LIN {X 0,Y 481.085,Z 509.859,A -85,B 0,C 180,E1 -6735.62,E2 -6735.62} C_VEL
LIN {X 0,Y 481.237,Z 504.412,A -85,B 0,C 180,E1 -6738.202,E2 -6738.202} C_VEL
LIN {X 0,Y 481.286,Z 497.171,A -85,B 0,C 180,E1 -6741.603,E2 -6741.603} C_VEL
LIN {X 0,Y 481.313,Z 491.765,A -85,B 0,C 180,E1 -6744.133,E2 -6744.133} C_VEL
LIN {X 0,Y 481.415,Z 488.11,A -85,B 0,C 180,E1 -6745.814,E2 -6745.814} C_VEL
LIN {X 0,Y 481.345,Z 485.341,A -85,B 0,C 180,E1 -6747.175,E2 -6747.175} C_VEL
LIN {X 0,Y 481.839,Z 485.279,A -85,B 0,C 180,E1 -6749.164,E2 -6749.164} C_VEL
LIN {X 0,Y 481.908,Z 485.27,A -85,B 0,C 180,E1 -6750.835,E2 -6750.835} C_VEL
LIN {X 0,Y 481.93,Z 485.268,A -85,B 0,C 180,E1 -6752.507,E2 -6752.507} C_VEL
LIN {X 0,Y 481.82,Z 485.281,A -85,B 0,C 180,E1 -6755.86,E2 -6755.86} C_VEL
LIN {X 0,Y 481.763,Z 485.289,A -85,B 0,C 180,E1 -6758.388,E2 -6758.388} C_VEL
LIN {X 0,Y 481.752,Z 485.289,A -85,B 0,C 180,E1 -6761.784,E2 -6761.784} C_VEL
LIN {X 0,Y 481.745,Z 485.289,A -85,B 0,C 180,E1 -6765.224,E2 -6765.224} C_VEL
LIN {X 0,Y 481.713,Z 485.294,A -85,B 0,C 180,E1 -6768.721,E2 -6768.721} C_VEL
LIN {X 0,Y 481.648,Z 485.301,A -85,B 0,C 180,E1 -6771.394,E2 -6771.394} C_VEL
LIN {X 0,Y 481.678,Z 485.301,A -85,B 0,C 180,E1 -6774.113,E2 -6774.113} C_VEL
LIN {X 0,Y 481.752,Z 485.288,A -85,B 0,C 180,E1 -6777.14,E2 -6777.14} C_VEL
LIN {X 0,Y 481.688,Z 485.297,A -85,B 0,C 180,E1 -6779.74,E2 -6779.74} C_VEL
LIN {X 0,Y 481.673,Z 485.299,A -85,B 0,C 180,E1 -6782.674,E2 -6782.674} C_VEL
LIN {X 0,Y 481.643,Z 485.303,A -85,B 0,C 180,E1 -6785.708,E2 -6785.708} C_VEL
LIN {X 0,Y 481.67,Z 485.298,A -85,B 0,C 180,E1 -6788.859,E2 -6788.859} C_VEL
LIN {X 0,Y 481.661,Z 485.303,A -85,B 0,C 180,E1 -6791.914,E2 -6791.914} C_VEL
LIN {X 0,Y 481.659,Z 485.301,A -85,B 0,C 180,E1 -6794.457,E2 -6794.457} C_VEL
LIN {X 0,Y 481.687,Z 485.297,A -85,B 0,C 180,E1 -6796.845,E2 -6796.845} C_VEL
LIN {X 0,Y 481.688,Z 485.3,A -85,B 0,C 180,E1 -6800.061,E2 -6800.061} C_VEL
LIN {X 0,Y 481.624,Z 485.304,A -85,B 0,C 180,E1 -6803.253,E2 -6803.253} C_VEL
LIN {X 0,Y 481.707,Z 485.295,A -85,B 0,C 180,E1 -6806.33,E2 -6806.33} C_VEL
LIN {X 0,Y 481.649,Z 485.302,A -85,B 0,C 180,E1 -6809.417,E2 -6809.417} C_VEL
LIN {X 0,Y 481.7,Z 485.297,A -85,B 0,C 180,E1 -6812.168,E2 -6812.168} C_VEL
LIN {X 0,Y 481.717,Z 485.292,A -85,B 0,C 180,E1 -6814.97,E2 -6814.97} C_VEL
LIN {X 0,Y 481.651,Z 485.303,A -85,B 0,C 180,E1 -6817.705,E2 -6817.705} C_VEL
LIN {X 0,Y 481.706,Z 485.295,A -85,B 0,C 180,E1 -6820.393,E2 -6820.393} C_VEL
LIN {X 0,Y 481.689,Z 485.297,A -85,B 0,C 180,E1 -6823.034,E2 -6823.034} C_VEL
LIN {X 0,Y 481.688,Z 485.298,A -85,B 0,C 180,E1 -6825.639,E2 -6825.639} C_VEL
LIN {X 0,Y 481.793,Z 485.286,A -85,B 0,C 180,E1 -6828.216,E2 -6828.216} C_VEL
LIN {X 0,Y 481.761,Z 485.289,A -85,B 0,C 180,E1 -6831.612,E2 -6831.612} C_VEL
LIN {X 0,Y 481.814,Z 485.283,A -85,B 0,C 180,E1 -6834.139,E2 -6834.139} C_VEL
LIN {X 0,Y 481.928,Z 485.268,A -85,B 0,C 180,E1 -6837.492,E2 -6837.492} C_VEL
LIN {X 0,Y 481.939,Z 485.267,A -85,B 0,C 180,E1 -6840,E2 -6840} C_VEL
LIN {X 0,Y 481.926,Z 485.268,A -85,B 0,C 180,E1 -6842.507,E2 -6842.507} C_VEL
LIN {X 0,Y 481.816,Z 485.283,A -85,B 0,C 180,E1 -6845.86,E2 -6845.86} C_VEL
LIN {X 0,Y 481.761,Z 485.289,A -85,B 0,C 180,E1 -6848.388,E2 -6848.388} C_VEL
LIN {X 0,Y 481.749,Z 485.291,A -85,B 0,C 180,E1 -6851.785,E2 -6851.785} C_VEL
LIN {X 0,Y 481.74,Z 485.291,A -85,B 0,C 180,E1 -6855.224,E2 -6855.224} C_VEL
LIN {X 0,Y 481.71,Z 485.293,A -85,B 0,C 180,E1 -6858.722,E2 -6858.722} C_VEL
LIN {X 0,Y 481.645,Z 485.304,A -85,B 0,C 180,E1 -6861.395,E2 -6861.395} C_VEL
LIN {X 0,Y 481.675,Z 485.299,A -85,B 0,C 180,E1 -6864.113,E2 -6864.113} C_VEL
LIN {X 0,Y 481.744,Z 485.29,A -85,B 0,C 180,E1 -6867.139,E2 -6867.139} C_VEL
LIN {X 0,Y 481.686,Z 485.3,A -85,B 0,C 180,E1 -6869.741,E2 -6869.741} C_VEL
LIN {X 0,Y 481.671,Z 485.299,A -85,B 0,C 180,E1 -6872.674,E2 -6872.674} C_VEL
LIN {X 0,Y 481.641,Z 485.306,A -85,B 0,C 180,E1 -6875.709,E2 -6875.709} C_VEL
LIN {X 0,Y 481.668,Z 485.299,A -85,B 0,C 180,E1 -6878.859,E2 -6878.859} C_VEL
LIN {X 0,Y 481.66,Z 485.301,A -85,B 0,C 180,E1 -6881.914,E2 -6881.914} C_VEL
LIN {X 0,Y 481.658,Z 485.3,A -85,B 0,C 180,E1 -6884.457,E2 -6884.457} C_VEL
LIN {X 0,Y 481.647,Z 485.303,A -85,B 0,C 180,E1 -6887.84,E2 -6887.84} C_VEL
LIN {X 0,Y 481.718,Z 485.292,A -85,B 0,C 180,E1 -6890.646,E2 -6890.646} C_VEL
LIN {X 0,Y 481.642,Z 485.305,A -85,B 0,C 180,E1 -6894.291,E2 -6894.291} C_VEL
LIN {X 0,Y 481.734,Z 485.411,A -85,B 0,C 180,E1 -6895.75,E2 -6895.75} C_VEL
LIN {X 0,Y 482.859,Z 492.268,A -85,B 0,C 180,E1 -6898.401,E2 -6898.401} C_VEL
LIN {X 0,Y 482.63,Z 499.151,A -85,B 0,C 180,E1 -6900.893,E2 -6900.893} C_VEL
LIN {X 0,Y 482.277,Z 506.878,A -85,B 0,C 180,E1 -6903.612,E2 -6903.612} C_VEL
LIN {X 0,Y 481.947,Z 514.883,A -85,B 0,C 180,E1 -6906.359,E2 -6906.359} C_VEL
LIN {X 0,Y 481.668,Z 524.244,A -85,B 0,C 180,E1 -6909.502,E2 -6909.502} C_VEL
LIN {X 0,Y 481.4,Z 533.634,A -85,B 0,C 180,E1 -6912.586,E2 -6912.586} C_VEL
LIN {X 0,Y 481.187,Z 543.054,A -85,B 0,C 180,E1 -6915.624,E2 -6915.624} C_VEL
LIN {X 0,Y 481.103,Z 551.174,A -85,B 0,C 180,E1 -6918.228,E2 -6918.228} C_VEL
LIN {X 0,Y 482.499,Z 564.801,A -85,B 0,C 180,E1 -6918.713,E2 -6918.713} C_VEL
LIN {X 0,Y 482.362,Z 574.583,A -85,B 0,C 180,E1 -6919.188,E2 -6919.188} C_VEL
LIN {X 0,Y 482.16,Z 583.023,A -85,B 0,C 180,E1 -6919.715,E2 -6919.715} C_VEL
LIN {X 0,Y 481.922,Z 591.176,A -85,B 0,C 180,E1 -6920.346,E2 -6920.346} C_VEL
LIN {X 0,Y 481.622,Z 598.943,A -85,B 0,C 180,E1 -6921.081,E2 -6921.081} C_VEL
LIN {X 0,Y 481.355,Z 607.096,A -85,B 0,C 180,E1 -6922.028,E2 -6922.028} C_VEL
LIN {X 0,Y 481.168,Z 614.279,A -85,B 0,C 180,E1 -6923.079,E2 -6923.079} C_VEL
LIN {X 0,Y 481.055,Z 619.93,A -85,B 0,C 180,E1 -6924.131,E2 -6924.131} C_VEL
LIN {X 0,Y 480.885,Z 625.177,A -85,B 0,C 180,E1 -6925.39,E2 -6925.39} C_VEL
LIN {X 0,Y 480.937,Z 627.877,A -85,B 0,C 180,E1 -6926.23,E2 -6926.23} C_VEL
LIN {X 0,Y 480.848,Z 630.817,A -85,B 0,C 180,E1 -6927.487,E2 -6927.487} C_VEL
LIN {X 0,Y 480.822,Z 632.089,A -85,B 0,C 180,E1 -6928.325,E2 -6928.325} C_VEL
LIN {X 0,Y 480.758,Z 632.873,A -85,B 0,C 180,E1 -6929.163,E2 -6929.163} C_VEL
LIN {X 0,Y 480.74,Z 633.154,A -85,B 0,C 180,E1 -6930,E2 -6930} C_VEL
LIN {X 0,Y 480.758,Z 632.838,A -85,B 0,C 180,E1 -6930.838,E2 -6930.838} C_VEL
LIN {X 0,Y 480.822,Z 632.029,A -85,B 0,C 180,E1 -6931.676,E2 -6931.676} C_VEL
LIN {X 0,Y 480.849,Z 630.732,A -85,B 0,C 180,E1 -6932.514,E2 -6932.514} C_VEL
LIN {X 0,Y 480.94,Z 627.734,A -85,B 0,C 180,E1 -6933.771,E2 -6933.771} C_VEL
LIN {X 0,Y 480.885,Z 624.999,A -85,B 0,C 180,E1 -6934.611,E2 -6934.611} C_VEL
LIN {X 0,Y 481.057,Z 619.674,A -85,B 0,C 180,E1 -6935.87,E2 -6935.87} C_VEL
LIN {X 0,Y 481.209,Z 612.625,A -85,B 0,C 180,E1 -6937.132,E2 -6937.132} C_VEL
LIN {X 0,Y 481.403,Z 604.966,A -85,B 0,C 180,E1 -6938.184,E2 -6938.184} C_VEL
LIN {X 0,Y 481.621,Z 598.453,A -85,B 0,C 180,E1 -6938.92,E2 -6938.92} C_VEL
LIN {X 0,Y 481.882,Z 590.591,A -85,B 0,C 180,E1 -6939.656,E2 -6939.656} C_VEL
LIN {X 0,Y 482.097,Z 582.346,A -85,B 0,C 180,E1 -6940.287,E2 -6940.287} C_VEL
LIN {X 0,Y 482.403,Z 571.991,A -85,B 0,C 180,E1 -6940.918,E2 -6940.918} C_VEL
LIN {X 0,Y 482.382,Z 564.502,A -85,B 0,C 180,E1 -6941.267,E2 -6941.267} C_VEL
LIN {X 0,Y 481.115,Z 552.246,A -85,B 0,C 180,E1 -6941.715,E2 -6941.715} C_VEL
LIN {X 0,Y 481.004,Z 550.841,A -85,B 0,C 180,E1 -6941.75,E2 -6941.75} C_VEL
LIN {X 0,Y 481.17,Z 540.308,A -85,B 0,C 180,E1 -6945.243,E2 -6945.243} C_VEL
LIN {X 0,Y 481.361,Z 530.012,A -85,B 0,C 180,E1 -6948.736,E2 -6948.736} C_VEL
LIN {X 0,Y 481.539,Z 521.127,A -85,B 0,C 180,E1 -6951.85,E2 -6951.85} C_VEL
LIN {X 0,Y 481.787,Z 513.681,A -85,B 0,C 180,E1 -6954.566,E2 -6954.566} C_VEL
LIN {X 0,Y 482.085,Z 506.773,A -85,B 0,C 180,E1 -6957.217,E2 -6957.217} C_VEL
LIN {X 0,Y 482.519,Z 499.627,A -85,B 0,C 180,E1 -6960.166,E2 -6960.166} C_VEL
LIN {X 0,Y 482.874,Z 494.307,A -85,B 0,C 180,E1 -6962.583,E2 -6962.583} C_VEL
LIN {X 0,Y 482.76,Z 491.673,A -85,B 0,C 180,E1 -6963.922,E2 -6963.922} C_VEL
LIN {X 0,Y 481.959,Z 486.988,A -85,B 0,C 180,E1 -6966.718,E2 -6966.718} C_VEL
LIN {X 0,Y 481.658,Z 485.303,A -85,B 0,C 180,E1 -6968.008,E2 -6968.008} C_VEL
LIN {X 0,Y 481.659,Z 485.302,A -85,B 0,C 180,E1 -6971.042,E2 -6971.042} C_VEL
LIN {X 0,Y 481.662,Z 485.301,A -85,B 0,C 180,E1 -6974.458,E2 -6974.458} C_VEL
LIN {X 0,Y 481.656,Z 485.302,A -85,B 0,C 180,E1 -6977.84,E2 -6977.84} C_VEL
LIN {X 0,Y 481.683,Z 485.299,A -85,B 0,C 180,E1 -6980.651,E2 -6980.651} C_VEL
LIN {X 0,Y 481.63,Z 485.307,A -85,B 0,C 180,E1 -6983.376,E2 -6983.376} C_VEL
LIN {X 0,Y 481.672,Z 485.303,A -85,B 0,C 180,E1 -6986.327,E2 -6986.327} C_VEL
LIN {X 0,Y 481.625,Z 485.502,A -85,B 0,C 180,E1 -6987.322,E2 -6987.322} C_VEL
LIN {X 0,Y 481.574,Z 488.341,A -85,B 0,C 180,E1 -6990.252,E2 -6990.252} C_VEL
LIN {X 0,Y 481.43,Z 491.329,A -85,B 0,C 180,E1 -6993.093,E2 -6993.093} C_VEL
LIN {X 0,Y 481.283,Z 494.419,A -85,B 0,C 180,E1 -6995.866,E2 -6995.866} C_VEL
LIN {X 0,Y 481.208,Z 498.618,A -85,B 0,C 180,E1 -6999.481,E2 -6999.481} C_VEL
LIN {X 0,Y 481.075,Z 501.825,A -85,B 0,C 180,E1 -7002.134,E2 -7002.134} C_VEL
LIN {X 0,Y 481.082,Z 505.064,A -85,B 0,C 180,E1 -7004.754,E2 -7004.754} C_VEL
LIN {X 0,Y 481.019,Z 509.748,A -85,B 0,C 180,E1 -7008.382,E2 -7008.382} C_VEL
LIN {X 0,Y 482.651,Z 519.951,A -85,B 0,C 180,E1 -7008.796,E2 -7008.796} C_VEL
LIN {X 0,Y 482.57,Z 529.986,A -85,B 0,C 180,E1 -7009.299,E2 -7009.299} C_VEL
LIN {X 0,Y 482.326,Z 538.199,A -85,B 0,C 180,E1 -7009.824,E2 -7009.824} C_VEL
LIN {X 0,Y 482.104,Z 546.171,A -85,B 0,C 180,E1 -7010.455,E2 -7010.455} C_VEL
LIN {X 0,Y 481.84,Z 553.789,A -85,B 0,C 180,E1 -7011.191,E2 -7011.191} C_VEL
LIN {X 0,Y 481.554,Z 562.569,A -85,B 0,C 180,E1 -7012.242,E2 -7012.242} C_VEL
LIN {X 0,Y 481.379,Z 569.346,A -85,B 0,C 180,E1 -7013.293,E2 -7013.293} C_VEL
LIN {X 0,Y 481.216,Z 573.822,A -85,B 0,C 180,E1 -7014.132,E2 -7014.132} C_VEL
LIN {X 0,Y 480.982,Z 577.55,A -85,B 0,C 180,E1 -7014.97,E2 -7014.97} C_VEL
LIN {X 0,Y 481.072,Z 580.556,A -85,B 0,C 180,E1 -7015.811,E2 -7015.811} C_VEL
LIN {X 0,Y 480.931,Z 582.902,A -85,B 0,C 180,E1 -7016.649,E2 -7016.649} C_VEL
LIN {X 0,Y 480.932,Z 584.693,A -85,B 0,C 180,E1 -7017.487,E2 -7017.487} C_VEL
LIN {X 0,Y 480.826,Z 585.985,A -85,B 0,C 180,E1 -7018.325,E2 -7018.325} C_VEL
LIN {X 0,Y 480.758,Z 586.796,A -85,B 0,C 180,E1 -7019.162,E2 -7019.162} C_VEL
LIN {X 0,Y 480.741,Z 587.086,A -85,B 0,C 180,E1 -7020,E2 -7020} C_VEL
LIN {X 0,Y 480.759,Z 586.792,A -85,B 0,C 180,E1 -7020.838,E2 -7020.838} C_VEL
LIN {X 0,Y 480.825,Z 586.022,A -85,B 0,C 180,E1 -7021.675,E2 -7021.675} C_VEL
LIN {X 0,Y 480.929,Z 584.774,A -85,B 0,C 180,E1 -7022.513,E2 -7022.513} C_VEL
LIN {X 0,Y 480.973,Z 581.859,A -85,B 0,C 180,E1 -7023.77,E2 -7023.77} C_VEL
LIN {X 0,Y 481.038,Z 579.21,A -85,B 0,C 180,E1 -7024.609,E2 -7024.609} C_VEL
LIN {X 0,Y 481.056,Z 575.944,A -85,B 0,C 180,E1 -7025.449,E2 -7025.449} C_VEL
LIN {X 0,Y 481.367,Z 570.596,A -85,B 0,C 180,E1 -7026.53,E2 -7026.53} C_VEL
LIN {X 0,Y 481.383,Z 565.894,A -85,B 0,C 180,E1 -7027.318,E2 -7027.318} C_VEL
LIN {X 0,Y 481.579,Z 559.676,A -85,B 0,C 180,E1 -7028.18,E2 -7028.18} C_VEL
LIN {X 0,Y 481.856,Z 552.295,A -85,B 0,C 180,E1 -7029.021,E2 -7029.021} C_VEL
LIN {X 0,Y 482.129,Z 544.414,A -85,B 0,C 180,E1 -7029.756,E2 -7029.756} C_VEL
LIN {X 0,Y 482.398,Z 534.626,A -85,B 0,C 180,E1 -7030.493,E2 -7030.493} C_VEL
LIN {X 0,Y 482.682,Z 523.618,A -85,B 0,C 180,E1 -7031.106,E2 -7031.106} C_VEL
LIN {X 0,Y 482.424,Z 518.253,A -85,B 0,C 180,E1 -7031.356,E2 -7031.356} C_VEL
LIN {X 0,Y 480.988,Z 508.57,A -85,B 0,C 180,E1 -7031.736,E2 -7031.736} C_VEL
LIN {X 0,Y 480.982,Z 503.343,A -85,B 0,C 180,E1 -7035.338,E2 -7035.338} C_VEL
LIN {X 0,Y 481.041,Z 498.477,A -85,B 0,C 180,E1 -7038.749,E2 -7038.749} C_VEL
LIN {X 0,Y 481.027,Z 494.705,A -85,B 0,C 180,E1 -7041.424,E2 -7041.424} C_VEL
LIN {X 0,Y 481.077,Z 490.923,A -85,B 0,C 180,E1 -7044.145,E2 -7044.145} C_VEL
LIN {X 0,Y 481.268,Z 486.758,A -85,B 0,C 180,E1 -7047.175,E2 -7047.175} C_VEL
LIN {X 0,Y 481.309,Z 492.917,A -85,B 0,C 180,E1 -7049.766,E2 -7049.766} C_VEL
LIN {X 0,Y 481.3,Z 499.781,A -85,B 0,C 180,E1 -7052.703,E2 -7052.703} C_VEL
LIN {X 0,Y 481.179,Z 506.791,A -85,B 0,C 180,E1 -7055.749,E2 -7055.749} C_VEL
LIN {X 0,Y 481.121,Z 513.978,A -85,B 0,C 180,E1 -7058.912,E2 -7058.912} C_VEL
LIN {X 0,Y 481.025,Z 521.479,A -85,B 0,C 180,E1 -7062.228,E2 -7062.228} C_VEL
LIN {X 0,Y 480.985,Z 526.164,A -85,B 0,C 180,E1 -7064.304,E2 -7064.304} C_VEL
LIN {X 0,Y 482.645,Z 537.384,A -85,B 0,C 180,E1 -7064.708,E2 -7064.708} C_VEL
LIN {X 0,Y 482.552,Z 549.204,A -85,B 0,C 180,E1 -7065.281,E2 -7065.281} C_VEL
LIN {X 0,Y 482.306,Z 556.838,A -85,B 0,C 180,E1 -7065.763,E2 -7065.763} C_VEL
LIN {X 0,Y 482.009,Z 565.549,A -85,B 0,C 180,E1 -7066.454,E2 -7066.454} C_VEL
LIN {X 0,Y 481.763,Z 572.859,A -85,B 0,C 180,E1 -7067.166,E2 -7067.166} C_VEL
LIN {X 0,Y 481.523,Z 579.942,A -85,B 0,C 180,E1 -7068.003,E2 -7068.003} C_VEL
LIN {X 0,Y 481.264,Z 586.293,A -85,B 0,C 180,E1 -7068.917,E2 -7068.917} C_VEL
LIN {X 0,Y 481.143,Z 592.383,A -85,B 0,C 180,E1 -7070.006,E2 -7070.006} C_VEL
LIN {X 0,Y 480.974,Z 597.017,A -85,B 0,C 180,E1 -7071.073,E2 -7071.073} C_VEL
LIN {X 0,Y 480.893,Z 600.561,A -85,B 0,C 180,E1 -7072.134,E2 -7072.134} C_VEL
LIN {X 0,Y 480.78,Z 603.774,A -85,B 0,C 180,E1 -7073.512,E2 -7073.512} C_VEL
LIN {X 0,Y 480.749,Z 605.7,A -85,B 0,C 180,E1 -7074.951,E2 -7074.951} C_VEL
LIN {X 0,Y 480.697,Z 605.997,A -85,B 0,C 180,E1 -7076.446,E2 -7076.446} C_VEL
LIN {X 0,Y 480.7,Z 605.58,A -85,B 0,C 180,E1 -7077.251,E2 -7077.251} C_VEL
LIN {X 0,Y 480.756,Z 604.566,A -85,B 0,C 180,E1 -7078.116,E2 -7078.116} C_VEL
LIN {X 0,Y 480.142,Z 603.435,A -85,B 0,C 180,E1 -7078.804,E2 -7078.804} C_VEL
LIN {X 0,Y 477.368,Z 600.944,A -85,B 0,C 180,E1 -7079.904,E2 -7079.904} C_VEL
LIN {X 0,Y 475.014,Z 598.301,A -85,B 0,C 180,E1 -7080.765,E2 -7080.765} C_VEL
LIN {X 0,Y 474.013,Z 595.889,A -85,B 0,C 180,E1 -7081.409,E2 -7081.409} C_VEL
LIN {X 0,Y 473.94,Z 594.965,A -85,B 0,C 180,E1 -7081.622,E2 -7081.622} C_VEL
LIN {X 0,Y 474.122,Z 590.034,A -85,B 0,C 180,E1 -7082.644,E2 -7082.644} C_VEL
LIN {X 0,Y 474.357,Z 584.27,A -85,B 0,C 180,E1 -7083.61,E2 -7083.61} C_VEL
LIN {X 0,Y 474.596,Z 577.044,A -85,B 0,C 180,E1 -7084.597,E2 -7084.597} C_VEL
LIN {X 0,Y 474.931,Z 568.471,A -85,B 0,C 180,E1 -7085.522,E2 -7085.522} C_VEL
LIN {X 0,Y 475.198,Z 560.21,A -85,B 0,C 180,E1 -7086.233,E2 -7086.233} C_VEL
LIN {X 0,Y 475.465,Z 551.667,A -85,B 0,C 180,E1 -7086.824,E2 -7086.824} C_VEL
LIN {X 0,Y 475.711,Z 543.001,A -85,B 0,C 180,E1 -7087.296,E2 -7087.296} C_VEL
LIN {X 0,Y 475.446,Z 537.02,A -85,B 0,C 180,E1 -7087.569,E2 -7087.569} C_VEL
LIN {X 0,Y 473.936,Z 527.336,A -85,B 0,C 180,E1 -7087.924,E2 -7087.924} C_VEL
LIN {X 0,Y 473.833,Z 526.451,A -85,B 0,C 180,E1 -7087.977,E2 -7087.977} C_VEL
LIN {X 0,Y 473.943,Z 518.809,A -85,B 0,C 180,E1 -7091.63,E2 -7091.63} C_VEL
LIN {X 0,Y 474.014,Z 512.776,A -85,B 0,C 180,E1 -7094.521,E2 -7094.521} C_VEL
LIN {X 0,Y 474.17,Z 505.433,A -85,B 0,C 180,E1 -7098.023,E2 -7098.023} C_VEL
LIN {X 0,Y 474.213,Z 498.134,A -85,B 0,C 180,E1 -7101.477,E2 -7101.477} C_VEL
LIN {X 0,Y 474.252,Z 492.69,A -85,B 0,C 180,E1 -7104.045,E2 -7104.045} C_VEL
LIN {X 0,Y 474.371,Z 489.028,A -85,B 0,C 180,E1 -7105.751,E2 -7105.751} C_VEL
LIN {X 0,Y 474.28,Z 486.222,A -85,B 0,C 180,E1 -7107.133,E2 -7107.133} C_VEL
LIN {X 0,Y 474.789,Z 486.157,A -85,B 0,C 180,E1 -7109.151,E2 -7109.151} C_VEL
LIN {X 0,Y 474.859,Z 486.148,A -85,B 0,C 180,E1 -7110.848,E2 -7110.848} C_VEL
LIN {X 0,Y 474.896,Z 486.145,A -85,B 0,C 180,E1 -7112.544,E2 -7112.544} C_VEL
LIN {X 0,Y 474.782,Z 486.158,A -85,B 0,C 180,E1 -7115.947,E2 -7115.947} C_VEL
LIN {X 0,Y 474.728,Z 486.166,A -85,B 0,C 180,E1 -7118.513,E2 -7118.513} C_VEL
LIN {X 0,Y 474.705,Z 486.167,A -85,B 0,C 180,E1 -7121.962,E2 -7121.962} C_VEL
LIN {X 0,Y 474.702,Z 486.166,A -85,B 0,C 180,E1 -7125.455,E2 -7125.455} C_VEL
LIN {X 0,Y 474.666,Z 486.172,A -85,B 0,C 180,E1 -7129.01,E2 -7129.01} C_VEL
LIN {X 0,Y 474.591,Z 486.182,A -85,B 0,C 180,E1 -7131.728,E2 -7131.728} C_VEL
LIN {X 0,Y 474.66,Z 486.173,A -85,B 0,C 180,E1 -7134.492,E2 -7134.492} C_VEL
LIN {X 0,Y 474.699,Z 486.166,A -85,B 0,C 180,E1 -7137.338,E2 -7137.338} C_VEL
LIN {X 0,Y 474.61,Z 486.179,A -85,B 0,C 180,E1 -7140.811,E2 -7140.811} C_VEL
LIN {X 0,Y 474.638,Z 486.177,A -85,B 0,C 180,E1 -7143.984,E2 -7143.984} C_VEL
LIN {X 0,Y 474.575,Z 486.184,A -85,B 0,C 180,E1 -7146.9,E2 -7146.9} C_VEL
LIN {X 0,Y 474.627,Z 486.179,A -85,B 0,C 180,E1 -7149.647,E2 -7149.647} C_VEL
LIN {X 0,Y 474.634,Z 486.176,A -85,B 0,C 180,E1 -7152.931,E2 -7152.931} C_VEL
LIN {X 0,Y 474.617,Z 486.179,A -85,B 0,C 180,E1 -7155.896,E2 -7155.896} C_VEL
LIN {X 0,Y 474.644,Z 486.175,A -85,B 0,C 180,E1 -7159.038,E2 -7159.038} C_VEL
LIN {X 0,Y 474.616,Z 486.18,A -85,B 0,C 180,E1 -7161.702,E2 -7161.702} C_VEL
LIN {X 0,Y 474.622,Z 486.178,A -85,B 0,C 180,E1 -7164.725,E2 -7164.725} C_VEL
LIN {X 0,Y 474.635,Z 486.177,A -85,B 0,C 180,E1 -7167.788,E2 -7167.788} C_VEL
LIN {X 0,Y 474.622,Z 486.177,A -85,B 0,C 180,E1 -7170.884,E2 -7170.884} C_VEL
LIN {X 0,Y 474.665,Z 486.173,A -85,B 0,C 180,E1 -7173.629,E2 -7173.629} C_VEL
LIN {X 0,Y 474.634,Z 486.177,A -85,B 0,C 180,E1 -7176.641,E2 -7176.641} C_VEL
LIN {X 0,Y 474.655,Z 486.176,A -85,B 0,C 180,E1 -7180.089,E2 -7180.089} C_VEL
LIN {X 0,Y 474.649,Z 486.174,A -85,B 0,C 180,E1 -7182.774,E2 -7182.774} C_VEL
LIN {X 0,Y 474.646,Z 486.175,A -85,B 0,C 180,E1 -7185.421,E2 -7185.421} C_VEL
LIN {X 0,Y 474.737,Z 486.164,A -85,B 0,C 180,E1 -7188.038,E2 -7188.038} C_VEL
LIN {X 0,Y 474.726,Z 486.165,A -85,B 0,C 180,E1 -7191.486,E2 -7191.486} C_VEL
LIN {X 0,Y 474.777,Z 486.159,A -85,B 0,C 180,E1 -7194.052,E2 -7194.052} C_VEL
LIN {X 0,Y 474.894,Z 486.144,A -85,B 0,C 180,E1 -7197.455,E2 -7197.455} C_VEL
LIN {X 0,Y 474.91,Z 486.143,A -85,B 0,C 180,E1 -7200,E2 -7200} C_VEL
LIN {X 0,Y 474.893,Z 486.144,A -85,B 0,C 180,E1 -7202.545,E2 -7202.545} C_VEL
LIN {X 0,Y 474.778,Z 486.16,A -85,B 0,C 180,E1 -7205.948,E2 -7205.948} C_VEL
LIN {X 0,Y 474.726,Z 486.165,A -85,B 0,C 180,E1 -7208.513,E2 -7208.513} C_VEL
LIN {X 0,Y 474.702,Z 486.17,A -85,B 0,C 180,E1 -7211.962,E2 -7211.962} C_VEL
LIN {X 0,Y 474.697,Z 486.169,A -85,B 0,C 180,E1 -7215.456,E2 -7215.456} C_VEL
LIN {X 0,Y 474.663,Z 486.172,A -85,B 0,C 180,E1 -7219.01,E2 -7219.01} C_VEL
LIN {X 0,Y 474.588,Z 486.184,A -85,B 0,C 180,E1 -7221.729,E2 -7221.729} C_VEL
LIN {X 0,Y 474.657,Z 486.172,A -85,B 0,C 180,E1 -7224.493,E2 -7224.493} C_VEL
LIN {X 0,Y 474.696,Z 486.169,A -85,B 0,C 180,E1 -7227.339,E2 -7227.339} C_VEL
LIN {X 0,Y 474.608,Z 486.178,A -85,B 0,C 180,E1 -7230.812,E2 -7230.812} C_VEL
LIN {X 0,Y 474.636,Z 486.176,A -85,B 0,C 180,E1 -7233.984,E2 -7233.984} C_VEL
LIN {X 0,Y 474.573,Z 486.184,A -85,B 0,C 180,E1 -7236.9,E2 -7236.9} C_VEL
LIN {X 0,Y 474.625,Z 486.178,A -85,B 0,C 180,E1 -7239.648,E2 -7239.648} C_VEL
LIN {X 0,Y 474.633,Z 486.177,A -85,B 0,C 180,E1 -7242.932,E2 -7242.932} C_VEL
LIN {X 0,Y 474.607,Z 486.18,A -85,B 0,C 180,E1 -7245.895,E2 -7245.895} C_VEL
LIN {X 0,Y 474.639,Z 486.177,A -85,B 0,C 180,E1 -7249.039,E2 -7249.039} C_VEL
LIN {X 0,Y 474.618,Z 486.179,A -85,B 0,C 180,E1 -7251.703,E2 -7251.703} C_VEL
LIN {X 0,Y 474.655,Z 486.175,A -85,B 0,C 180,E1 -7255.247,E2 -7255.247} C_VEL
LIN {X 0,Y 474.667,Z 486.306,A -85,B 0,C 180,E1 -7255.57,E2 -7255.57} C_VEL
LIN {X 0,Y 475.875,Z 493.46,A -85,B 0,C 180,E1 -7258.38,E2 -7258.38} C_VEL
LIN {X 0,Y 475.626,Z 500.087,A -85,B 0,C 180,E1 -7260.816,E2 -7260.816} C_VEL
LIN {X 0,Y 475.252,Z 508.062,A -85,B 0,C 180,E1 -7263.664,E2 -7263.664} C_VEL
LIN {X 0,Y 474.885,Z 516.406,A -85,B 0,C 180,E1 -7266.572,E2 -7266.572} C_VEL
LIN {X 0,Y 474.591,Z 525.398,A -85,B 0,C 180,E1 -7269.635,E2 -7269.635} C_VEL
LIN {X 0,Y 474.296,Z 534.759,A -85,B 0,C 180,E1 -7272.762,E2 -7272.762} C_VEL
LIN {X 0,Y 474.078,Z 544.139,A -85,B 0,C 180,E1 -7275.842,E2 -7275.842} C_VEL
LIN {X 0,Y 474.019,Z 550.954,A -85,B 0,C 180,E1 -7278.06,E2 -7278.06} C_VEL
LIN {X 0,Y 475.437,Z 564.436,A -85,B 0,C 180,E1 -7278.547,E2 -7278.547} C_VEL
LIN {X 0,Y 475.354,Z 574.134,A -85,B 0,C 180,E1 -7279.027,E2 -7279.027} C_VEL
LIN {X 0,Y 475.168,Z 582.592,A -85,B 0,C 180,E1 -7279.562,E2 -7279.562} C_VEL
LIN {X 0,Y 474.881,Z 590.757,A -85,B 0,C 180,E1 -7280.201,E2 -7280.201} C_VEL
LIN {X 0,Y 474.596,Z 598.54,A -85,B 0,C 180,E1 -7280.948,E2 -7280.948} C_VEL
LIN {X 0,Y 474.347,Z 604.995,A -85,B 0,C 180,E1 -7281.695,E2 -7281.695} C_VEL
LIN {X 0,Y 474.145,Z 611.157,A -85,B 0,C 180,E1 -7282.548,E2 -7282.548} C_VEL
LIN {X 0,Y 473.992,Z 616.408,A -85,B 0,C 180,E1 -7283.426,E2 -7283.426} C_VEL
LIN {X 0,Y 473.929,Z 621.501,A -85,B 0,C 180,E1 -7284.469,E2 -7284.469} C_VEL
LIN {X 0,Y 473.779,Z 626.335,A -85,B 0,C 180,E1 -7285.747,E2 -7285.747} C_VEL
LIN {X 0,Y 473.848,Z 628.697,A -85,B 0,C 180,E1 -7286.599,E2 -7286.599} C_VEL
LIN {X 0,Y 473.765,Z 630.478,A -85,B 0,C 180,E1 -7287.45,E2 -7287.45} C_VEL
LIN {X 0,Y 473.755,Z 631.753,A -85,B 0,C 180,E1 -7288.3,E2 -7288.3} C_VEL
LIN {X 0,Y 473.686,Z 632.538,A -85,B 0,C 180,E1 -7289.15,E2 -7289.15} C_VEL
LIN {X 0,Y 473.666,Z 632.816,A -85,B 0,C 180,E1 -7290,E2 -7290} C_VEL
LIN {X 0,Y 473.686,Z 632.496,A -85,B 0,C 180,E1 -7290.851,E2 -7290.851} C_VEL
LIN {X 0,Y 473.755,Z 631.68,A -85,B 0,C 180,E1 -7291.701,E2 -7291.701} C_VEL
LIN {X 0,Y 473.766,Z 630.371,A -85,B 0,C 180,E1 -7292.551,E2 -7292.551} C_VEL
LIN {X 0,Y 473.844,Z 627.361,A -85,B 0,C 180,E1 -7293.827,E2 -7293.827} C_VEL
LIN {X 0,Y 473.806,Z 624.612,A -85,B 0,C 180,E1 -7294.68,E2 -7294.68} C_VEL
LIN {X 0,Y 473.965,Z 619.27,A -85,B 0,C 180,E1 -7295.958,E2 -7295.958} C_VEL
LIN {X 0,Y 474.126,Z 612.201,A -85,B 0,C 180,E1 -7297.239,E2 -7297.239} C_VEL
LIN {X 0,Y 474.289,Z 606.259,A -85,B 0,C 180,E1 -7298.093,E2 -7298.093} C_VEL
LIN {X 0,Y 474.551,Z 599.047,A -85,B 0,C 180,E1 -7298.946,E2 -7298.946} C_VEL
LIN {X 0,Y 474.829,Z 591.391,A -85,B 0,C 180,E1 -7299.693,E2 -7299.693} C_VEL
LIN {X 0,Y 475.042,Z 583.41,A -85,B 0,C 180,E1 -7300.334,E2 -7300.334} C_VEL
LIN {X 0,Y 475.302,Z 575.25,A -85,B 0,C 180,E1 -7300.867,E2 -7300.867} C_VEL
LIN {X 0,Y 475.462,Z 566.183,A -85,B 0,C 180,E1 -7301.337,E2 -7301.337} C_VEL
LIN {X 0,Y 474.473,Z 556.197,A -85,B 0,C 180,E1 -7301.751,E2 -7301.751} C_VEL
LIN {X 0,Y 473.936,Z 550.451,A -85,B 0,C 180,E1 -7301.934,E2 -7301.934} C_VEL
LIN {X 0,Y 474.086,Z 539.884,A -85,B 0,C 180,E1 -7305.511,E2 -7305.511} C_VEL
LIN {X 0,Y 474.298,Z 529.755,A -85,B 0,C 180,E1 -7309.026,E2 -7309.026} C_VEL
LIN {X 0,Y 474.512,Z 520.935,A -85,B 0,C 180,E1 -7312.19,E2 -7312.19} C_VEL
LIN {X 0,Y 474.788,Z 513.57,A -85,B 0,C 180,E1 -7314.953,E2 -7314.953} C_VEL
LIN {X 0,Y 475.235,Z 505.335,A -85,B 0,C 180,E1 -7318.245,E2 -7318.245} C_VEL
LIN {X 0,Y 475.684,Z 498.694,A -85,B 0,C 180,E1 -7321.139,E2 -7321.139} C_VEL
LIN {X 0,Y 475.923,Z 494.6,A -85,B 0,C 180,E1 -7323.12,E2 -7323.12} C_VEL
LIN {X 0,Y 475.321,Z 490.255,A -85,B 0,C 180,E1 -7325.589,E2 -7325.589} C_VEL
LIN {X 0,Y 474.614,Z 486.213,A -85,B 0,C 180,E1 -7328.458,E2 -7328.458} C_VEL
LIN {X 0,Y 474.63,Z 486.178,A -85,B 0,C 180,E1 -7330.96,E2 -7330.96} C_VEL
LIN {X 0,Y 474.612,Z 486.179,A -85,B 0,C 180,E1 -7334.105,E2 -7334.105} C_VEL
LIN {X 0,Y 474.638,Z 486.177,A -85,B 0,C 180,E1 -7337.068,E2 -7337.068} C_VEL
LIN {X 0,Y 474.647,Z 486.175,A -85,B 0,C 180,E1 -7340.454,E2 -7340.454} C_VEL
LIN {X 0,Y 474.591,Z 486.183,A -85,B 0,C 180,E1 -7343.677,E2 -7343.677} C_VEL
LIN {X 0,Y 474.578,Z 486.189,A -85,B 0,C 180,E1 -7346.775,E2 -7346.775} C_VEL
LIN {X 0,Y 474.613,Z 488.358,A -85,B 0,C 180,E1 -7349.189,E2 -7349.189} C_VEL
LIN {X 0,Y 474.455,Z 490.858,A -85,B 0,C 180,E1 -7351.705,E2 -7351.705} C_VEL
LIN {X 0,Y 474.312,Z 493.99,A -85,B 0,C 180,E1 -7354.67,E2 -7354.67} C_VEL
LIN {X 0,Y 474.172,Z 496.967,A -85,B 0,C 180,E1 -7357.334,E2 -7357.334} C_VEL
LIN {X 0,Y 474.089,Z 500.115,A -85,B 0,C 180,E1 -7360.065,E2 -7360.065} C_VEL
LIN {X 0,Y 473.973,Z 503.328,A -85,B 0,C 180,E1 -7362.749,E2 -7362.749} C_VEL
LIN {X 0,Y 473.969,Z 506.579,A -85,B 0,C 180,E1 -7365.4,E2 -7365.4} C_VEL
LIN {X 0,Y 473.959,Z 510.105,A -85,B 0,C 180,E1 -7368.204,E2 -7368.204} C_VEL
LIN {X 0,Y 475.757,Z 521.268,A -85,B 0,C 180,E1 -7368.675,E2 -7368.675} C_VEL
LIN {X 0,Y 475.623,Z 530.335,A -85,B 0,C 180,E1 -7369.141,E2 -7369.141} C_VEL
LIN {X 0,Y 475.358,Z 538.539,A -85,B 0,C 180,E1 -7369.673,E2 -7369.673} C_VEL
LIN {X 0,Y 475.116,Z 546.51,A -85,B 0,C 180,E1 -7370.313,E2 -7370.313} C_VEL
LIN {X 0,Y 474.849,Z 554.128,A -85,B 0,C 180,E1 -7371.06,E2 -7371.06} C_VEL
LIN {X 0,Y 474.531,Z 562.916,A -85,B 0,C 180,E1 -7372.126,E2 -7372.126} C_VEL
LIN {X 0,Y 474.331,Z 569.699,A -85,B 0,C 180,E1 -7373.193,E2 -7373.193} C_VEL
LIN {X 0,Y 474.18,Z 574.172,A -85,B 0,C 180,E1 -7374.045,E2 -7374.045} C_VEL
LIN {X 0,Y 473.916,Z 577.902,A -85,B 0,C 180,E1 -7374.895,E2 -7374.895} C_VEL
LIN {X 0,Y 474.014,Z 580.904,A -85,B 0,C 180,E1 -7375.749,E2 -7375.749} C_VEL
LIN {X 0,Y 473.865,Z 583.25,A -85,B 0,C 180,E1 -7376.599,E2 -7376.599} C_VEL
LIN {X 0,Y 473.855,Z 585.04,A -85,B 0,C 180,E1 -7377.45,E2 -7377.45} C_VEL
LIN {X 0,Y 473.761,Z 586.331,A -85,B 0,C 180,E1 -7378.3,E2 -7378.3} C_VEL
LIN {X 0,Y 473.687,Z 587.139,A -85,B 0,C 180,E1 -7379.15,E2 -7379.15} C_VEL
LIN {X 0,Y 473.668,Z 587.427,A -85,B 0,C 180,E1 -7380,E2 -7380} C_VEL
LIN {X 0,Y 473.688,Z 587.128,A -85,B 0,C 180,E1 -7380.85,E2 -7380.85} C_VEL
LIN {X 0,Y 473.76,Z 586.35,A -85,B 0,C 180,E1 -7381.7,E2 -7381.7} C_VEL
LIN {X 0,Y 473.838,Z 585.093,A -85,B 0,C 180,E1 -7382.55,E2 -7382.55} C_VEL
LIN {X 0,Y 473.912,Z 582.166,A -85,B 0,C 180,E1 -7383.826,E2 -7383.826} C_VEL
LIN {X 0,Y 473.955,Z 579.505,A -85,B 0,C 180,E1 -7384.678,E2 -7384.678} C_VEL
LIN {X 0,Y 474.01,Z 576.222,A -85,B 0,C 180,E1 -7385.53,E2 -7385.53} C_VEL
LIN {X 0,Y 474.328,Z 570.894,A -85,B 0,C 180,E1 -7386.622,E2 -7386.622} C_VEL
LIN {X 0,Y 474.344,Z 566.138,A -85,B 0,C 180,E1 -7387.428,E2 -7387.428} C_VEL
LIN {X 0,Y 474.567,Z 559.9,A -85,B 0,C 180,E1 -7388.302,E2 -7388.302} C_VEL
LIN {X 0,Y 474.861,Z 552.499,A -85,B 0,C 180,E1 -7389.155,E2 -7389.155} C_VEL
LIN {X 0,Y 475.123,Z 544.597,A -85,B 0,C 180,E1 -7389.902,E2 -7389.902} C_VEL
LIN {X 0,Y 475.423,Z 534.782,A -85,B 0,C 180,E1 -7390.649,E2 -7390.649} C_VEL
LIN {X 0,Y 475.72,Z 524.364,A -85,B 0,C 180,E1 -7391.241,E2 -7391.241} C_VEL
LIN {X 0,Y 475.353,Z 517.924,A -85,B 0,C 180,E1 -7391.545,E2 -7391.545} C_VEL
LIN {X 0,Y 473.923,Z 508.858,A -85,B 0,C 180,E1 -7391.904,E2 -7391.904} C_VEL
LIN {X 0,Y 473.9,Z 503.699,A -85,B 0,C 180,E1 -7395.482,E2 -7395.482} C_VEL
LIN {X 0,Y 473.963,Z 498.655,A -85,B 0,C 180,E1 -7399.04,E2 -7399.04} C_VEL
LIN {X 0,Y 473.95,Z 494.858,A -85,B 0,C 180,E1 -7401.76,E2 -7401.76} C_VEL
LIN {X 0,Y 474.028,Z 491.038,A -85,B 0,C 180,E1 -7404.528,E2 -7404.528} C_VEL
LIN {X 0,Y 474.226,Z 487.481,A -85,B 0,C 180,E1 -7407.143,E2 -7407.143} C_VEL
LIN {X 0,Y 474.24,Z 493.623,A -85,B 0,C 180,E1 -7409.766,E2 -7409.766} C_VEL
LIN {X 0,Y 474.249,Z 500.634,A -85,B 0,C 180,E1 -7412.77,E2 -7412.77} C_VEL
LIN {X 0,Y 474.103,Z 507.69,A -85,B 0,C 180,E1 -7415.842,E2 -7415.842} C_VEL
LIN {X 0,Y 474.068,Z 514.882,A -85,B 0,C 180,E1 -7419.033,E2 -7419.033} C_VEL
LIN {X 0,Y 473.944,Z 521.884,A -85,B 0,C 180,E1 -7422.145,E2 -7422.145} C_VEL
LIN {X 0,Y 473.906,Z 526.342,A -85,B 0,C 180,E1 -7424.134,E2 -7424.134} C_VEL
LIN {X 0,Y 475.433,Z 536.183,A -85,B 0,C 180,E1 -7424.484,E2 -7424.484} C_VEL
LIN {X 0,Y 475.707,Z 541.927,A -85,B 0,C 180,E1 -7424.735,E2 -7424.735} C_VEL
LIN {X 0,Y 475.482,Z 551.529,A -85,B 0,C 180,E1 -7425.25,E2 -7425.25} C_VEL
LIN {X 0,Y 475.215,Z 559.792,A -85,B 0,C 180,E1 -7425.818,E2 -7425.818} C_VEL
LIN {X 0,Y 474.912,Z 568.931,A -85,B 0,C 180,E1 -7426.602,E2 -7426.602} C_VEL
LIN {X 0,Y 474.603,Z 576.853,A -85,B 0,C 180,E1 -7427.458,E2 -7427.458} C_VEL
LIN {X 0,Y 474.328,Z 584.062,A -85,B 0,C 180,E1 -7428.436,E2 -7428.436} C_VEL
LIN {X 0,Y 474.145,Z 589.278,A -85,B 0,C 180,E1 -7429.293,E2 -7429.293} C_VEL
LIN {X 0,Y 473.977,Z 594.658,A -85,B 0,C 180,E1 -7430.387,E2 -7430.387} C_VEL
LIN {X 0,Y 473.849,Z 598.834,A -85,B 0,C 180,E1 -7431.469,E2 -7431.469} C_VEL
LIN {X 0,Y 473.775,Z 601.974,A -85,B 0,C 180,E1 -7432.54,E2 -7432.54} C_VEL
LIN {X 0,Y 473.702,Z 604.191,A -85,B 0,C 180,E1 -7433.597,E2 -7433.597} C_VEL
LIN {X 0,Y 473.663,Z 605.637,A -85,B 0,C 180,E1 -7434.693,E2 -7434.693} C_VEL
LIN {X 0,Y 473.624,Z 606.281,A -85,B 0,C 180,E1 -7436.199,E2 -7436.199} C_VEL
LIN {X 0,Y 473.65,Z 605.23,A -85,B 0,C 180,E1 -7437.754,E2 -7437.754} C_VEL
LIN {X 0,Y 473.789,Z 602.456,A -85,B 0,C 180,E1 -7439.356,E2 -7439.356} C_VEL
LIN {X 0,Y 473.809,Z 600.202,A -85,B 0,C 180,E1 -7440.204,E2 -7440.204} C_VEL
LIN {X 0,Y 473.936,Z 596.113,A -85,B 0,C 180,E1 -7441.359,E2 -7441.359} C_VEL
LIN {X 0,Y 473.94,Z 594.965,A -85,B 0,C 180,E1 -7441.622,E2 -7441.622} C_VEL
LIN {X 0,Y 473.333,Z 592.221,A -85,B 0,C 180,E1 -7442.247,E2 -7442.247} C_VEL
LIN {X 0,Y 470.677,Z 587.118,A -85,B 0,C 180,E1 -7443.235,E2 -7443.235} C_VEL
LIN {X 0,Y 468.08,Z 581.365,A -85,B 0,C 180,E1 -7444.17,E2 -7444.17} C_VEL
LIN {X 0,Y 467.567,Z 577.374,A -85,B 0,C 180,E1 -7444.702,E2 -7444.702} C_VEL
LIN {X 0,Y 467.948,Z 567.973,A -85,B 0,C 180,E1 -7445.723,E2 -7445.723} C_VEL
LIN {X 0,Y 468.217,Z 560.19,A -85,B 0,C 180,E1 -7446.397,E2 -7446.397} C_VEL
LIN {X 0,Y 468.471,Z 552.61,A -85,B 0,C 180,E1 -7446.935,E2 -7446.935} C_VEL
LIN {X 0,Y 468.749,Z 543.124,A -85,B 0,C 180,E1 -7447.464,E2 -7447.464} C_VEL
LIN {X 0,Y 468.434,Z 537.242,A -85,B 0,C 180,E1 -7447.738,E2 -7447.738} C_VEL
LIN {X 0,Y 466.743,Z 526.617,A -85,B 0,C 180,E1 -7448.148,E2 -7448.148} C_VEL
LIN {X 0,Y 466.865,Z 519.507,A -85,B 0,C 180,E1 -7451.571,E2 -7451.571} C_VEL
LIN {X 0,Y 466.953,Z 512.013,A -85,B 0,C 180,E1 -7455.175,E2 -7455.175} C_VEL
LIN {X 0,Y 467.115,Z 504.624,A -85,B 0,C 180,E1 -7458.72,E2 -7458.72} C_VEL
LIN {X 0,Y 467.168,Z 497.29,A -85,B 0,C 180,E1 -7462.218,E2 -7462.218} C_VEL
LIN {X 0,Y 467.327,Z 489.926,A -85,B 0,C 180,E1 -7465.687,E2 -7465.687} C_VEL
LIN {X 0,Y 467.234,Z 487.1,A -85,B 0,C 180,E1 -7467.09,E2 -7467.09} C_VEL
LIN {X 0,Y 467.741,Z 487.035,A -85,B 0,C 180,E1 -7469.139,E2 -7469.139} C_VEL
LIN {X 0,Y 467.812,Z 487.026,A -85,B 0,C 180,E1 -7470.86,E2 -7470.86} C_VEL
LIN {X 0,Y 467.861,Z 487.021,A -85,B 0,C 180,E1 -7472.582,E2 -7472.582} C_VEL
LIN {X 0,Y 467.747,Z 487.034,A -85,B 0,C 180,E1 -7476.037,E2 -7476.037} C_VEL
LIN {X 0,Y 467.682,Z 487.044,A -85,B 0,C 180,E1 -7478.642,E2 -7478.642} C_VEL
LIN {X 0,Y 467.657,Z 487.046,A -85,B 0,C 180,E1 -7482.145,E2 -7482.145} C_VEL
LIN {X 0,Y 467.64,Z 487.047,A -85,B 0,C 180,E1 -7485.694,E2 -7485.694} C_VEL
LIN {X 0,Y 467.619,Z 487.05,A -85,B 0,C 180,E1 -7488.764,E2 -7488.764} C_VEL
LIN {X 0,Y 467.582,Z 487.052,A -85,B 0,C 180,E1 -7491.268,E2 -7491.268} C_VEL
LIN {X 0,Y 467.574,Z 487.056,A -85,B 0,C 180,E1 -7493.943,E2 -7493.943} C_VEL
LIN {X 0,Y 467.628,Z 487.048,A -85,B 0,C 180,E1 -7496.799,E2 -7496.799} C_VEL
LIN {X 0,Y 467.587,Z 487.054,A -85,B 0,C 180,E1 -7499.735,E2 -7499.735} C_VEL
LIN {X 0,Y 467.583,Z 487.053,A -85,B 0,C 180,E1 -7502.758,E2 -7502.758} C_VEL
LIN {X 0,Y 467.556,Z 487.059,A -85,B 0,C 180,E1 -7505.889,E2 -7505.889} C_VEL
LIN {X 0,Y 467.581,Z 487.053,A -85,B 0,C 180,E1 -7509.144,E2 -7509.144} C_VEL
LIN {X 0,Y 467.585,Z 487.055,A -85,B 0,C 180,E1 -7512.567,E2 -7512.567} C_VEL
LIN {X 0,Y 467.569,Z 487.055,A -85,B 0,C 180,E1 -7515.053,E2 -7515.053} C_VEL
LIN {X 0,Y 467.623,Z 487.049,A -85,B 0,C 180,E1 -7517.444,E2 -7517.444} C_VEL
LIN {X 0,Y 467.614,Z 487.05,A -85,B 0,C 180,E1 -7520.858,E2 -7520.858} C_VEL
LIN {X 0,Y 467.557,Z 487.058,A -85,B 0,C 180,E1 -7524.261,E2 -7524.261} C_VEL
LIN {X 0,Y 467.58,Z 487.055,A -85,B 0,C 180,E1 -7527.32,E2 -7527.32} C_VEL
LIN {X 0,Y 467.568,Z 487.057,A -85,B 0,C 180,E1 -7530.667,E2 -7530.667} C_VEL
LIN {X 0,Y 467.626,Z 487.049,A -85,B 0,C 180,E1 -7533.2,E2 -7533.2} C_VEL
LIN {X 0,Y 467.591,Z 487.055,A -85,B 0,C 180,E1 -7536.468,E2 -7536.468} C_VEL
LIN {X 0,Y 467.622,Z 487.05,A -85,B 0,C 180,E1 -7539.777,E2 -7539.777} C_VEL
LIN {X 0,Y 467.607,Z 487.052,A -85,B 0,C 180,E1 -7542.507,E2 -7542.507} C_VEL
LIN {X 0,Y 467.604,Z 487.052,A -85,B 0,C 180,E1 -7545.196,E2 -7545.196} C_VEL
LIN {X 0,Y 467.681,Z 487.043,A -85,B 0,C 180,E1 -7547.855,E2 -7547.855} C_VEL
LIN {X 0,Y 467.68,Z 487.043,A -85,B 0,C 180,E1 -7551.357,E2 -7551.357} C_VEL
LIN {X 0,Y 467.741,Z 487.036,A -85,B 0,C 180,E1 -7553.963,E2 -7553.963} C_VEL
LIN {X 0,Y 467.859,Z 487.02,A -85,B 0,C 180,E1 -7557.417,E2 -7557.417} C_VEL
LIN {X 0,Y 467.88,Z 487.019,A -85,B 0,C 180,E1 -7560,E2 -7560} C_VEL
LIN {X 0,Y 467.858,Z 487.02,A -85,B 0,C 180,E1 -7562.583,E2 -7562.583} C_VEL
LIN {X 0,Y 467.742,Z 487.037,A -85,B 0,C 180,E1 -7566.037,E2 -7566.037} C_VEL
LIN {X 0,Y 467.68,Z 487.042,A -85,B 0,C 180,E1 -7568.643,E2 -7568.643} C_VEL
LIN {X 0,Y 467.653,Z 487.046,A -85,B 0,C 180,E1 -7572.145,E2 -7572.145} C_VEL
LIN {X 0,Y 467.637,Z 487.05,A -85,B 0,C 180,E1 -7575.695,E2 -7575.695} C_VEL
LIN {X 0,Y 467.615,Z 487.048,A -85,B 0,C 180,E1 -7578.765,E2 -7578.765} C_VEL
LIN {X 0,Y 467.578,Z 487.055,A -85,B 0,C 180,E1 -7581.269,E2 -7581.269} C_VEL
LIN {X 0,Y 467.571,Z 487.057,A -85,B 0,C 180,E1 -7583.943,E2 -7583.943} C_VEL
LIN {X 0,Y 467.614,Z 487.05,A -85,B 0,C 180,E1 -7586.8,E2 -7586.8} C_VEL
LIN {X 0,Y 467.585,Z 487.057,A -85,B 0,C 180,E1 -7589.736,E2 -7589.736} C_VEL
LIN {X 0,Y 467.581,Z 487.054,A -85,B 0,C 180,E1 -7592.758,E2 -7592.758} C_VEL
LIN {X 0,Y 467.554,Z 487.059,A -85,B 0,C 180,E1 -7595.889,E2 -7595.889} C_VEL
LIN {X 0,Y 467.579,Z 487.055,A -85,B 0,C 180,E1 -7599.145,E2 -7599.145} C_VEL
LIN {X 0,Y 467.584,Z 487.053,A -85,B 0,C 180,E1 -7602.567,E2 -7602.567} C_VEL
LIN {X 0,Y 467.568,Z 487.056,A -85,B 0,C 180,E1 -7605.053,E2 -7605.053} C_VEL
LIN {X 0,Y 467.586,Z 487.056,A -85,B 0,C 180,E1 -7607.44,E2 -7607.44} C_VEL
LIN {X 0,Y 467.617,Z 487.049,A -85,B 0,C 180,E1 -7610.859,E2 -7610.859} C_VEL
LIN {X 0,Y 467.562,Z 487.058,A -85,B 0,C 180,E1 -7614.261,E2 -7614.261} C_VEL
LIN {X 0,Y 467.644,Z 487.251,A -85,B 0,C 180,E1 -7615.412,E2 -7615.412} C_VEL
LIN {X 0,Y 468.695,Z 493.304,A -85,B 0,C 180,E1 -7617.838,E2 -7617.838} C_VEL
LIN {X 0,Y 468.842,Z 497.286,A -85,B 0,C 180,E1 -7619.359,E2 -7619.359} C_VEL
LIN {X 0,Y 468.402,Z 505.236,A -85,B 0,C 180,E1 -7622.282,E2 -7622.282} C_VEL
LIN {X 0,Y 468.028,Z 513.209,A -85,B 0,C 180,E1 -7625.137,E2 -7625.137} C_VEL
LIN {X 0,Y 467.635,Z 522.472,A -85,B 0,C 180,E1 -7628.378,E2 -7628.378} C_VEL
LIN {X 0,Y 467.33,Z 531.125,A -85,B 0,C 180,E1 -7631.34,E2 -7631.34} C_VEL
LIN {X 0,Y 467.089,Z 541.303,A -85,B 0,C 180,E1 -7634.763,E2 -7634.763} C_VEL
LIN {X 0,Y 466.938,Z 550.767,A -85,B 0,C 180,E1 -7637.9,E2 -7637.9} C_VEL
LIN {X 0,Y 468.101,Z 562.479,A -85,B 0,C 180,E1 -7638.305,E2 -7638.305} C_VEL
LIN {X 0,Y 468.52,Z 568.586,A -85,B 0,C 180,E1 -7638.596,E2 -7638.596} C_VEL
LIN {X 0,Y 468.247,Z 579.078,A -85,B 0,C 180,E1 -7639.187,E2 -7639.187} C_VEL
LIN {X 0,Y 467.875,Z 589.073,A -85,B 0,C 180,E1 -7639.944,E2 -7639.944} C_VEL
LIN {X 0,Y 467.54,Z 597.08,A -85,B 0,C 180,E1 -7640.701,E2 -7640.701} C_VEL
LIN {X 0,Y 467.371,Z 602.87,A -85,B 0,C 180,E1 -7641.352,E2 -7641.352} C_VEL
LIN {X 0,Y 467.114,Z 609.331,A -85,B 0,C 180,E1 -7642.218,E2 -7642.218} C_VEL
LIN {X 0,Y 467.001,Z 614.714,A -85,B 0,C 180,E1 -7643.086,E2 -7643.086} C_VEL
LIN {X 0,Y 466.868,Z 619.203,A -85,B 0,C 180,E1 -7643.952,E2 -7643.952} C_VEL
LIN {X 0,Y 466.809,Z 622.941,A -85,B 0,C 180,E1 -7644.818,E2 -7644.818} C_VEL
LIN {X 0,Y 466.689,Z 625.982,A -85,B 0,C 180,E1 -7645.682,E2 -7645.682} C_VEL
LIN {X 0,Y 466.761,Z 628.349,A -85,B 0,C 180,E1 -7646.548,E2 -7646.548} C_VEL
LIN {X 0,Y 466.685,Z 630.136,A -85,B 0,C 180,E1 -7647.411,E2 -7647.411} C_VEL
LIN {X 0,Y 466.66,Z 631.413,A -85,B 0,C 180,E1 -7648.274,E2 -7648.274} C_VEL
LIN {X 0,Y 466.618,Z 632.199,A -85,B 0,C 180,E1 -7649.137,E2 -7649.137} C_VEL
LIN {X 0,Y 466.596,Z 632.478,A -85,B 0,C 180,E1 -7650,E2 -7650} C_VEL
LIN {X 0,Y 466.618,Z 632.156,A -85,B 0,C 180,E1 -7650.863,E2 -7650.863} C_VEL
LIN {X 0,Y 466.66,Z 631.335,A -85,B 0,C 180,E1 -7651.726,E2 -7651.726} C_VEL
LIN {X 0,Y 466.686,Z 630.022,A -85,B 0,C 180,E1 -7652.59,E2 -7652.59} C_VEL
LIN {X 0,Y 466.734,Z 627.004,A -85,B 0,C 180,E1 -7653.886,E2 -7653.886} C_VEL
LIN {X 0,Y 466.732,Z 624.251,A -85,B 0,C 180,E1 -7654.751,E2 -7654.751} C_VEL
LIN {X 0,Y 466.852,Z 620.866,A -85,B 0,C 180,E1 -7655.616,E2 -7655.616} C_VEL
LIN {X 0,Y 466.941,Z 616.108,A -85,B 0,C 180,E1 -7656.599,E2 -7656.599} C_VEL
LIN {X 0,Y 467.069,Z 610.366,A -85,B 0,C 180,E1 -7657.566,E2 -7657.566} C_VEL
LIN {X 0,Y 467.297,Z 604.131,A -85,B 0,C 180,E1 -7658.433,E2 -7658.433} C_VEL
LIN {X 0,Y 467.478,Z 597.597,A -85,B 0,C 180,E1 -7659.192,E2 -7659.192} C_VEL
LIN {X 0,Y 467.768,Z 590.963,A -85,B 0,C 180,E1 -7659.841,E2 -7659.841} C_VEL
LIN {X 0,Y 468.048,Z 582.981,A -85,B 0,C 180,E1 -7660.49,E2 -7660.49} C_VEL
LIN {X 0,Y 468.33,Z 574.829,A -85,B 0,C 180,E1 -7661.031,E2 -7661.031} C_VEL
LIN {X 0,Y 468.46,Z 566.691,A -85,B 0,C 180,E1 -7661.467,E2 -7661.467} C_VEL
LIN {X 0,Y 467.594,Z 557.519,A -85,B 0,C 180,E1 -7661.869,E2 -7661.869} C_VEL
LIN {X 0,Y 466.841,Z 550.028,A -85,B 0,C 180,E1 -7662.141,E2 -7662.141} C_VEL
LIN {X 0,Y 467,Z 540.004,A -85,B 0,C 180,E1 -7665.603,E2 -7665.603} C_VEL
LIN {X 0,Y 467.197,Z 531.491,A -85,B 0,C 180,E1 -7668.612,E2 -7668.612} C_VEL
LIN {X 0,Y 467.392,Z 523.246,A -85,B 0,C 180,E1 -7671.617,E2 -7671.617} C_VEL
LIN {X 0,Y 467.692,Z 515.901,A -85,B 0,C 180,E1 -7674.409,E2 -7674.409} C_VEL
LIN {X 0,Y 468.04,Z 508.914,A -85,B 0,C 180,E1 -7677.211,E2 -7677.211} C_VEL
LIN {X 0,Y 468.515,Z 502.089,A -85,B 0,C 180,E1 -7680.167,E2 -7680.167} C_VEL
LIN {X 0,Y 468.931,Z 496.882,A -85,B 0,C 180,E1 -7682.653,E2 -7682.653} C_VEL
LIN {X 0,Y 468.615,Z 493.115,A -85,B 0,C 180,E1 -7684.744,E2 -7684.744} C_VEL
LIN {X 0,Y 467.963,Z 489.342,A -85,B 0,C 180,E1 -7687.253,E2 -7687.253} C_VEL
LIN {X 0,Y 467.569,Z 487.059,A -85,B 0,C 180,E1 -7689.147,E2 -7689.147} C_VEL
LIN {X 0,Y 467.589,Z 487.054,A -85,B 0,C 180,E1 -7692.567,E2 -7692.567} C_VEL
LIN {X 0,Y 467.573,Z 487.057,A -85,B 0,C 180,E1 -7695.053,E2 -7695.053} C_VEL
LIN {X 0,Y 467.591,Z 487.054,A -85,B 0,C 180,E1 -7697.44,E2 -7697.44} C_VEL
LIN {X 0,Y 467.585,Z 487.056,A -85,B 0,C 180,E1 -7700.856,E2 -7700.856} C_VEL
LIN {X 0,Y 467.562,Z 487.059,A -85,B 0,C 180,E1 -7704.261,E2 -7704.261} C_VEL
LIN {X 0,Y 467.559,Z 487.06,A -85,B 0,C 180,E1 -7706.21,E2 -7706.21} C_VEL
LIN {X 0,Y 467.625,Z 488.634,A -85,B 0,C 180,E1 -7708.263,E2 -7708.263} C_VEL
LIN {X 0,Y 467.461,Z 491.423,A -85,B 0,C 180,E1 -7711.243,E2 -7711.243} C_VEL
LIN {X 0,Y 467.287,Z 494.737,A -85,B 0,C 180,E1 -7714.476,E2 -7714.476} C_VEL
LIN {X 0,Y 467.091,Z 498.478,A -85,B 0,C 180,E1 -7717.904,E2 -7717.904} C_VEL
LIN {X 0,Y 467.002,Z 501.64,A -85,B 0,C 180,E1 -7720.666,E2 -7720.666} C_VEL
LIN {X 0,Y 466.943,Z 506.095,A -85,B 0,C 180,E1 -7724.424,E2 -7724.424} C_VEL
LIN {X 0,Y 466.892,Z 510.516,A -85,B 0,C 180,E1 -7728.003,E2 -7728.003} C_VEL
LIN {X 0,Y 468.708,Z 521.149,A -85,B 0,C 180,E1 -7728.471,E2 -7728.471} C_VEL
LIN {X 0,Y 468.683,Z 530.755,A -85,B 0,C 180,E1 -7728.978,E2 -7728.978} C_VEL
LIN {X 0,Y 468.396,Z 538.906,A -85,B 0,C 180,E1 -7729.518,E2 -7729.518} C_VEL
LIN {X 0,Y 468.139,Z 546.843,A -85,B 0,C 180,E1 -7730.168,E2 -7730.168} C_VEL
LIN {X 0,Y 467.849,Z 554.467,A -85,B 0,C 180,E1 -7730.925,E2 -7730.925} C_VEL
LIN {X 0,Y 467.51,Z 563.263,A -85,B 0,C 180,E1 -7732.007,E2 -7732.007} C_VEL
LIN {X 0,Y 467.285,Z 570.052,A -85,B 0,C 180,E1 -7733.089,E2 -7733.089} C_VEL
LIN {X 0,Y 467.146,Z 574.528,A -85,B 0,C 180,E1 -7733.955,E2 -7733.955} C_VEL
LIN {X 0,Y 466.855,Z 578.26,A -85,B 0,C 180,E1 -7734.818,E2 -7734.818} C_VEL
LIN {X 0,Y 466.957,Z 581.263,A -85,B 0,C 180,E1 -7735.684,E2 -7735.684} C_VEL
LIN {X 0,Y 466.802,Z 583.61,A -85,B 0,C 180,E1 -7736.547,E2 -7736.547} C_VEL
LIN {X 0,Y 466.768,Z 585.399,A -85,B 0,C 180,E1 -7737.411,E2 -7737.411} C_VEL
LIN {X 0,Y 466.698,Z 586.685,A -85,B 0,C 180,E1 -7738.274,E2 -7738.274} C_VEL
LIN {X 0,Y 466.619,Z 587.488,A -85,B 0,C 180,E1 -7739.137,E2 -7739.137} C_VEL
LIN {X 0,Y 466.597,Z 587.771,A -85,B 0,C 180,E1 -7740,E2 -7740} C_VEL
LIN {X 0,Y 466.62,Z 587.465,A -85,B 0,C 180,E1 -7740.863,E2 -7740.863} C_VEL
LIN {X 0,Y 466.697,Z 586.677,A -85,B 0,C 180,E1 -7741.726,E2 -7741.726} C_VEL
LIN {X 0,Y 466.752,Z 585.406,A -85,B 0,C 180,E1 -7742.589,E2 -7742.589} C_VEL
LIN {X 0,Y 466.854,Z 582.46,A -85,B 0,C 180,E1 -7743.884,E2 -7743.884} C_VEL
LIN {X 0,Y 466.88,Z 579.78,A -85,B 0,C 180,E1 -7744.749,E2 -7744.749} C_VEL
LIN {X 0,Y 466.968,Z 576.474,A -85,B 0,C 180,E1 -7745.614,E2 -7745.614} C_VEL
LIN {X 0,Y 467.282,Z 571.501,A -85,B 0,C 180,E1 -7746.652,E2 -7746.652} C_VEL
LIN {X 0,Y 467.319,Z 566.196,A -85,B 0,C 180,E1 -7747.562,E2 -7747.562} C_VEL
LIN {X 0,Y 467.547,Z 560.072,A -85,B 0,C 180,E1 -7748.428,E2 -7748.428} C_VEL
LIN {X 0,Y 467.848,Z 552.638,A -85,B 0,C 180,E1 -7749.293,E2 -7749.293} C_VEL
LIN {X 0,Y 468.142,Z 544.7,A -85,B 0,C 180,E1 -7750.051,E2 -7750.051} C_VEL
LIN {X 0,Y 468.468,Z 534.84,A -85,B 0,C 180,E1 -7750.809,E2 -7750.809} C_VEL
LIN {X 0,Y 468.766,Z 523.376,A -85,B 0,C 180,E1 -7751.454,E2 -7751.454} C_VEL
LIN {X 0,Y 467.932,Z 515.572,A -85,B 0,C 180,E1 -7751.813,E2 -7751.813} C_VEL
LIN {X 0,Y 466.826,Z 509.141,A -85,B 0,C 180,E1 -7752.08,E2 -7752.08} C_VEL
LIN {X 0,Y 466.811,Z 503.923,A -85,B 0,C 180,E1 -7755.724,E2 -7755.724} C_VEL
LIN {X 0,Y 466.88,Z 500.019,A -85,B 0,C 180,E1 -7758.495,E2 -7758.495} C_VEL
LIN {X 0,Y 466.897,Z 496.286,A -85,B 0,C 180,E1 -7761.178,E2 -7761.178} C_VEL
LIN {X 0,Y 466.947,Z 492.454,A -85,B 0,C 180,E1 -7763.977,E2 -7763.977} C_VEL
LIN {X 0,Y 467.157,Z 488.259,A -85,B 0,C 180,E1 -7767.113,E2 -7767.113} C_VEL
LIN {X 0,Y 467.198,Z 494.426,A -85,B 0,C 180,E1 -7769.763,E2 -7769.763} C_VEL
LIN {X 0,Y 467.186,Z 501.403,A -85,B 0,C 180,E1 -7772.79,E2 -7772.79} C_VEL
LIN {X 0,Y 467.037,Z 508.581,A -85,B 0,C 180,E1 -7775.936,E2 -7775.936} C_VEL
LIN {X 0,Y 466.986,Z 515.926,A -85,B 0,C 180,E1 -7779.204,E2 -7779.204} C_VEL
LIN {X 0,Y 466.867,Z 523.581,A -85,B 0,C 180,E1 -7782.642,E2 -7782.642} C_VEL
LIN {X 0,Y 466.825,Z 526.482,A -85,B 0,C 180,E1 -7783.943,E2 -7783.943} C_VEL
LIN {X 0,Y 468.509,Z 537.209,A -85,B 0,C 180,E1 -7784.342,E2 -7784.342} C_VEL
LIN {X 0,Y 468.743,Z 543.046,A -85,B 0,C 180,E1 -7784.611,E2 -7784.611} C_VEL
LIN {X 0,Y 468.551,Z 551.507,A -85,B 0,C 180,E1 -7785.076,E2 -7785.076} C_VEL
LIN {X 0,Y 468.244,Z 560.131,A -85,B 0,C 180,E1 -7785.676,E2 -7785.676} C_VEL
LIN {X 0,Y 467.893,Z 568.953,A -85,B 0,C 180,E1 -7786.443,E2 -7786.443} C_VEL
LIN {X 0,Y 467.563,Z 577.863,A -85,B 0,C 180,E1 -7787.436,E2 -7787.436} C_VEL
LIN {X 0,Y 467.301,Z 583.987,A -85,B 0,C 180,E1 -7788.279,E2 -7788.279} C_VEL
LIN {X 0,Y 467.08,Z 589.679,A -85,B 0,C 180,E1 -7789.23,E2 -7789.23} C_VEL
LIN {X 0,Y 466.936,Z 594.162,A -85,B 0,C 180,E1 -7790.141,E2 -7790.141} C_VEL
LIN {X 0,Y 466.801,Z 598.312,A -85,B 0,C 180,E1 -7791.19,E2 -7791.19} C_VEL
LIN {X 0,Y 466.735,Z 600.58,A -85,B 0,C 180,E1 -7791.875,E2 -7791.875} C_VEL
LIN {X 0,Y 466.664,Z 603.287,A -85,B 0,C 180,E1 -7792.957,E2 -7792.957} C_VEL
LIN {X 0,Y 466.563,Z 605.569,A -85,B 0,C 180,E1 -7794.432,E2 -7794.432} C_VEL
LIN {X 0,Y 466.537,Z 606.184,A -85,B 0,C 180,E1 -7795.079,E2 -7795.079} C_VEL
LIN {X 0,Y 466.525,Z 606.496,A -85,B 0,C 180,E1 -7796.124,E2 -7796.124} C_VEL
LIN {X 0,Y 466.54,Z 605.701,A -85,B 0,C 180,E1 -7797.521,E2 -7797.521} C_VEL
LIN {X 0,Y 466.575,Z 604.959,A -85,B 0,C 180,E1 -7798.183,E2 -7798.183} C_VEL
LIN {X 0,Y 466.674,Z 603.118,A -85,B 0,C 180,E1 -7799.2,E2 -7799.2} C_VEL
LIN {X 0,Y 466.765,Z 599.431,A -85,B 0,C 180,E1 -7800.557,E2 -7800.557} C_VEL
LIN {X 0,Y 466.878,Z 595.19,A -85,B 0,C 180,E1 -7801.694,E2 -7801.694} C_VEL
LIN {X 0,Y 467.058,Z 590.969,A -85,B 0,C 180,E1 -7802.598,E2 -7802.598} C_VEL
LIN {X 0,Y 467.228,Z 586.39,A -85,B 0,C 180,E1 -7803.416,E2 -7803.416} C_VEL
LIN {X 0,Y 467.465,Z 579.455,A -85,B 0,C 180,E1 -7804.43,E2 -7804.43} C_VEL
LIN {X 0,Y 467.567,Z 577.374,A -85,B 0,C 180,E1 -7804.702,E2 -7804.702} C_VEL
LIN {X 0,Y 467.062,Z 573.169,A -85,B 0,C 180,E1 -7805.21,E2 -7805.21} C_VEL
LIN {X 0,Y 464.527,Z 566.04,A -85,B 0,C 180,E1 -7806.002,E2 -7806.002} C_VEL
LIN {X 0,Y 462.003,Z 558.336,A -85,B 0,C 180,E1 -7806.706,E2 -7806.706} C_VEL
LIN {X 0,Y 461.506,Z 553.236,A -85,B 0,C 180,E1 -7807.069,E2 -7807.069} C_VEL
LIN {X 0,Y 461.764,Z 544.47,A -85,B 0,C 180,E1 -7807.576,E2 -7807.576} C_VEL
LIN {X 0,Y 461.562,Z 538.735,A -85,B 0,C 180,E1 -7807.86,E2 -7807.86} C_VEL
LIN {X 0,Y 459.863,Z 528.036,A -85,B 0,C 180,E1 -7808.276,E2 -7808.276} C_VEL
LIN {X 0,Y 459.665,Z 526.721,A -85,B 0,C 180,E1 -7808.354,E2 -7808.354} C_VEL
LIN {X 0,Y 459.759,Z 520.437,A -85,B 0,C 180,E1 -7811.397,E2 -7811.397} C_VEL
LIN {X 0,Y 459.865,Z 513.132,A -85,B 0,C 180,E1 -7814.941,E2 -7814.941} C_VEL
LIN {X 0,Y 460.032,Z 505.692,A -85,B 0,C 180,E1 -7818.544,E2 -7818.544} C_VEL
LIN {X 0,Y 460.093,Z 498.255,A -85,B 0,C 180,E1 -7822.098,E2 -7822.098} C_VEL
LIN {X 0,Y 460.285,Z 490.856,A -85,B 0,C 180,E1 -7825.621,E2 -7825.621} C_VEL
LIN {X 0,Y 460.188,Z 487.978,A -85,B 0,C 180,E1 -7827.045,E2 -7827.045} C_VEL
LIN {X 0,Y 460.695,Z 487.912,A -85,B 0,C 180,E1 -7829.125,E2 -7829.125} C_VEL
LIN {X 0,Y 460.764,Z 487.903,A -85,B 0,C 180,E1 -7830.874,E2 -7830.874} C_VEL
LIN {X 0,Y 460.826,Z 487.898,A -85,B 0,C 180,E1 -7832.622,E2 -7832.622} C_VEL
LIN {X 0,Y 460.713,Z 487.911,A -85,B 0,C 180,E1 -7836.129,E2 -7836.129} C_VEL
LIN {X 0,Y 460.629,Z 487.921,A -85,B 0,C 180,E1 -7838.776,E2 -7838.776} C_VEL
LIN {X 0,Y 460.614,Z 487.924,A -85,B 0,C 180,E1 -7842.444,E2 -7842.444} C_VEL
LIN {X 0,Y 460.601,Z 487.926,A -85,B 0,C 180,E1 -7845.997,E2 -7845.997} C_VEL
LIN {X 0,Y 460.572,Z 487.927,A -85,B 0,C 180,E1 -7848.902,E2 -7848.902} C_VEL
LIN {X 0,Y 460.516,Z 487.933,A -85,B 0,C 180,E1 -7851.485,E2 -7851.485} C_VEL
LIN {X 0,Y 460.543,Z 487.933,A -85,B 0,C 180,E1 -7854.332,E2 -7854.332} C_VEL
LIN {X 0,Y 460.584,Z 487.924,A -85,B 0,C 180,E1 -7857.243,E2 -7857.243} C_VEL
LIN {X 0,Y 460.527,Z 487.935,A -85,B 0,C 180,E1 -7860.238,E2 -7860.238} C_VEL
LIN {X 0,Y 460.529,Z 487.932,A -85,B 0,C 180,E1 -7863.324,E2 -7863.324} C_VEL
LIN {X 0,Y 460.478,Z 487.94,A -85,B 0,C 180,E1 -7866.529,E2 -7866.529} C_VEL
LIN {X 0,Y 460.557,Z 487.931,A -85,B 0,C 180,E1 -7869.859,E2 -7869.859} C_VEL
LIN {X 0,Y 460.515,Z 487.935,A -85,B 0,C 180,E1 -7872.9,E2 -7872.9} C_VEL
LIN {X 0,Y 460.522,Z 487.935,A -85,B 0,C 180,E1 -7875.828,E2 -7875.828} C_VEL
LIN {X 0,Y 460.541,Z 487.931,A -85,B 0,C 180,E1 -7878.99,E2 -7878.99} C_VEL
LIN {X 0,Y 460.543,Z 487.931,A -85,B 0,C 180,E1 -7881.269,E2 -7881.269} C_VEL
LIN {X 0,Y 460.508,Z 487.937,A -85,B 0,C 180,E1 -7884.554,E2 -7884.554} C_VEL
LIN {X 0,Y 460.53,Z 487.934,A -85,B 0,C 180,E1 -7887.715,E2 -7887.715} C_VEL
LIN {X 0,Y 460.538,Z 487.932,A -85,B 0,C 180,E1 -7890.769,E2 -7890.769} C_VEL
LIN {X 0,Y 460.566,Z 487.929,A -85,B 0,C 180,E1 -7893.735,E2 -7893.735} C_VEL
LIN {X 0,Y 460.544,Z 487.931,A -85,B 0,C 180,E1 -7896.624,E2 -7896.624} C_VEL
LIN {X 0,Y 460.55,Z 487.931,A -85,B 0,C 180,E1 -7899.453,E2 -7899.453} C_VEL
LIN {X 0,Y 460.557,Z 487.931,A -85,B 0,C 180,E1 -7902.23,E2 -7902.23} C_VEL
LIN {X 0,Y 460.563,Z 487.928,A -85,B 0,C 180,E1 -7904.965,E2 -7904.965} C_VEL
LIN {X 0,Y 460.627,Z 487.922,A -85,B 0,C 180,E1 -7907.666,E2 -7907.666} C_VEL
LIN {X 0,Y 460.627,Z 487.922,A -85,B 0,C 180,E1 -7911.224,E2 -7911.224} C_VEL
LIN {X 0,Y 460.707,Z 487.912,A -85,B 0,C 180,E1 -7913.87,E2 -7913.87} C_VEL
LIN {X 0,Y 460.824,Z 487.897,A -85,B 0,C 180,E1 -7917.378,E2 -7917.378} C_VEL
LIN {X 0,Y 460.851,Z 487.894,A -85,B 0,C 180,E1 -7920,E2 -7920} C_VEL
LIN {X 0,Y 460.823,Z 487.896,A -85,B 0,C 180,E1 -7922.622,E2 -7922.622} C_VEL
LIN {X 0,Y 460.708,Z 487.912,A -85,B 0,C 180,E1 -7926.13,E2 -7926.13} C_VEL
LIN {X 0,Y 460.627,Z 487.92,A -85,B 0,C 180,E1 -7928.776,E2 -7928.776} C_VEL
LIN {X 0,Y 460.61,Z 487.921,A -85,B 0,C 180,E1 -7932.445,E2 -7932.445} C_VEL
LIN {X 0,Y 460.597,Z 487.925,A -85,B 0,C 180,E1 -7935.998,E2 -7935.998} C_VEL
LIN {X 0,Y 460.569,Z 487.926,A -85,B 0,C 180,E1 -7938.902,E2 -7938.902} C_VEL
LIN {X 0,Y 460.513,Z 487.937,A -85,B 0,C 180,E1 -7941.486,E2 -7941.486} C_VEL
LIN {X 0,Y 460.54,Z 487.93,A -85,B 0,C 180,E1 -7944.332,E2 -7944.332} C_VEL
LIN {X 0,Y 460.577,Z 487.927,A -85,B 0,C 180,E1 -7947.243,E2 -7947.243} C_VEL
LIN {X 0,Y 460.525,Z 487.932,A -85,B 0,C 180,E1 -7950.239,E2 -7950.239} C_VEL
LIN {X 0,Y 460.527,Z 487.935,A -85,B 0,C 180,E1 -7953.325,E2 -7953.325} C_VEL
LIN {X 0,Y 460.476,Z 487.938,A -85,B 0,C 180,E1 -7956.529,E2 -7956.529} C_VEL
LIN {X 0,Y 460.542,Z 487.93,A -85,B 0,C 180,E1 -7958.898,E2 -7958.898} C_VEL
LIN {X 0,Y 460.521,Z 487.933,A -85,B 0,C 180,E1 -7962.182,E2 -7962.182} C_VEL
LIN {X 0,Y 460.515,Z 487.937,A -85,B 0,C 180,E1 -7965.412,E2 -7965.412} C_VEL
LIN {X 0,Y 460.533,Z 487.932,A -85,B 0,C 180,E1 -7968.397,E2 -7968.397} C_VEL
LIN {X 0,Y 460.546,Z 487.933,A -85,B 0,C 180,E1 -7971.27,E2 -7971.27} C_VEL
LIN {X 0,Y 460.569,Z 487.93,A -85,B 0,C 180,E1 -7975.054,E2 -7975.054} C_VEL
LIN {X 0,Y 460.771,Z 489.136,A -85,B 0,C 180,E1 -7975.643,E2 -7975.643} C_VEL
LIN {X 0,Y 461.714,Z 494.462,A -85,B 0,C 180,E1 -7977.809,E2 -7977.809} C_VEL
LIN {X 0,Y 461.84,Z 498.44,A -85,B 0,C 180,E1 -7979.351,E2 -7979.351} C_VEL
LIN {X 0,Y 461.351,Z 506.703,A -85,B 0,C 180,E1 -7982.433,E2 -7982.433} C_VEL
LIN {X 0,Y 460.976,Z 514.345,A -85,B 0,C 180,E1 -7985.212,E2 -7985.212} C_VEL
LIN {X 0,Y 460.583,Z 523.758,A -85,B 0,C 180,E1 -7988.559,E2 -7988.559} C_VEL
LIN {X 0,Y 460.244,Z 532.953,A -85,B 0,C 180,E1 -7991.758,E2 -7991.758} C_VEL
LIN {X 0,Y 459.981,Z 542.286,A -85,B 0,C 180,E1 -7994.946,E2 -7994.946} C_VEL
LIN {X 0,Y 459.848,Z 550.469,A -85,B 0,C 180,E1 -7997.717,E2 -7997.717} C_VEL
LIN {X 0,Y 461.088,Z 562.559,A -85,B 0,C 180,E1 -7998.155,E2 -7998.155} C_VEL
LIN {X 0,Y 461.496,Z 569.885,A -85,B 0,C 180,E1 -7998.513,E2 -7998.513} C_VEL
LIN {X 0,Y 461.213,Z 580.09,A -85,B 0,C 180,E1 -7999.131,E2 -7999.131} C_VEL
LIN {X 0,Y 460.849,Z 588.568,A -85,B 0,C 180,E1 -7999.789,E2 -7999.789} C_VEL
LIN {X 0,Y 460.524,Z 596.602,A -85,B 0,C 180,E1 -8000.558,E2 -8000.558} C_VEL
LIN {X 0,Y 460.31,Z 602.412,A -85,B 0,C 180,E1 -8001.218,E2 -8001.218} C_VEL
LIN {X 0,Y 460.07,Z 608.896,A -85,B 0,C 180,E1 -8002.098,E2 -8002.098} C_VEL
LIN {X 0,Y 459.94,Z 614.298,A -85,B 0,C 180,E1 -8002.979,E2 -8002.979} C_VEL
LIN {X 0,Y 459.777,Z 618.803,A -85,B 0,C 180,E1 -8003.858,E2 -8003.858} C_VEL
LIN {X 0,Y 459.722,Z 622.558,A -85,B 0,C 180,E1 -8004.738,E2 -8004.738} C_VEL
LIN {X 0,Y 459.626,Z 626.814,A -85,B 0,C 180,E1 -8006.055,E2 -8006.055} C_VEL
LIN {X 0,Y 459.609,Z 629.78,A -85,B 0,C 180,E1 -8007.371,E2 -8007.371} C_VEL
LIN {X 0,Y 459.569,Z 631.065,A -85,B 0,C 180,E1 -8008.248,E2 -8008.248} C_VEL
LIN {X 0,Y 459.551,Z 631.859,A -85,B 0,C 180,E1 -8009.124,E2 -8009.124} C_VEL
LIN {X 0,Y 459.527,Z 632.137,A -85,B 0,C 180,E1 -8010,E2 -8010} C_VEL
LIN {X 0,Y 459.551,Z 631.815,A -85,B 0,C 180,E1 -8010.877,E2 -8010.877} C_VEL
LIN {X 0,Y 459.57,Z 630.995,A -85,B 0,C 180,E1 -8011.753,E2 -8011.753} C_VEL
LIN {X 0,Y 459.609,Z 629.68,A -85,B 0,C 180,E1 -8012.63,E2 -8012.63} C_VEL
LIN {X 0,Y 459.628,Z 626.651,A -85,B 0,C 180,E1 -8013.946,E2 -8013.946} C_VEL
LIN {X 0,Y 459.662,Z 623.895,A -85,B 0,C 180,E1 -8014.824,E2 -8014.824} C_VEL
LIN {X 0,Y 459.787,Z 618.523,A -85,B 0,C 180,E1 -8016.143,E2 -8016.143} C_VEL
LIN {X 0,Y 459.978,Z 611.42,A -85,B 0,C 180,E1 -8017.463,E2 -8017.463} C_VEL
LIN {X 0,Y 460.185,Z 605.454,A -85,B 0,C 180,E1 -8018.343,E2 -8018.343} C_VEL
LIN {X 0,Y 460.453,Z 597.196,A -85,B 0,C 180,E1 -8019.333,E2 -8019.333} C_VEL
LIN {X 0,Y 460.724,Z 590.588,A -85,B 0,C 180,E1 -8019.993,E2 -8019.993} C_VEL
LIN {X 0,Y 461.053,Z 582.655,A -85,B 0,C 180,E1 -8020.651,E2 -8020.651} C_VEL
LIN {X 0,Y 461.35,Z 574.573,A -85,B 0,C 180,E1 -8021.2,E2 -8021.2} C_VEL
LIN {X 0,Y 461.453,Z 567.171,A -85,B 0,C 180,E1 -8021.613,E2 -8021.613} C_VEL
LIN {X 0,Y 460.597,Z 558.051,A -85,B 0,C 180,E1 -8022.035,E2 -8022.035} C_VEL
LIN {X 0,Y 459.735,Z 549.619,A -85,B 0,C 180,E1 -8022.358,E2 -8022.358} C_VEL
LIN {X 0,Y 459.936,Z 540.121,A -85,B 0,C 180,E1 -8025.706,E2 -8025.706} C_VEL
LIN {X 0,Y 460.141,Z 530.669,A -85,B 0,C 180,E1 -8029.125,E2 -8029.125} C_VEL
LIN {X 0,Y 460.369,Z 523.088,A -85,B 0,C 180,E1 -8031.964,E2 -8031.964} C_VEL
LIN {X 0,Y 460.688,Z 515.834,A -85,B 0,C 180,E1 -8034.805,E2 -8034.805} C_VEL
LIN {X 0,Y 461.102,Z 508.459,A -85,B 0,C 180,E1 -8037.869,E2 -8037.869} C_VEL
LIN {X 0,Y 461.607,Z 502.256,A -85,B 0,C 180,E1 -8040.667,E2 -8040.667} C_VEL
LIN {X 0,Y 461.912,Z 499.166,A -85,B 0,C 180,E1 -8042.177,E2 -8042.177} C_VEL
LIN {X 0,Y 461.771,Z 495.346,A -85,B 0,C 180,E1 -8044.273,E2 -8044.273} C_VEL
LIN {X 0,Y 461.226,Z 491.955,A -85,B 0,C 180,E1 -8046.461,E2 -8046.461} C_VEL
LIN {X 0,Y 460.698,Z 488.848,A -85,B 0,C 180,E1 -8048.921,E2 -8048.921} C_VEL
LIN {X 0,Y 460.533,Z 487.935,A -85,B 0,C 180,E1 -8049.863,E2 -8049.863} C_VEL
LIN {X 0,Y 460.516,Z 487.936,A -85,B 0,C 180,E1 -8052.901,E2 -8052.901} C_VEL
LIN {X 0,Y 460.522,Z 487.934,A -85,B 0,C 180,E1 -8055.83,E2 -8055.83} C_VEL
LIN {X 0,Y 460.536,Z 487.933,A -85,B 0,C 180,E1 -8058.989,E2 -8058.989} C_VEL
LIN {X 0,Y 460.529,Z 487.935,A -85,B 0,C 180,E1 -8061.267,E2 -8061.267} C_VEL
LIN {X 0,Y 460.511,Z 487.937,A -85,B 0,C 180,E1 -8064.554,E2 -8064.554} C_VEL
LIN {X 0,Y 460.539,Z 487.934,A -85,B 0,C 180,E1 -8065.623,E2 -8065.623} C_VEL
LIN {X 0,Y 460.626,Z 489.342,A -85,B 0,C 180,E1 -8067.723,E2 -8067.723} C_VEL
LIN {X 0,Y 460.494,Z 492.03,A -85,B 0,C 180,E1 -8070.766,E2 -8070.766} C_VEL
LIN {X 0,Y 460.27,Z 495.497,A -85,B 0,C 180,E1 -8074.276,E2 -8074.276} C_VEL
LIN {X 0,Y 460.057,Z 498.977,A -85,B 0,C 180,E1 -8077.548,E2 -8077.548} C_VEL
LIN {X 0,Y 459.97,Z 502.105,A -85,B 0,C 180,E1 -8080.358,E2 -8080.358} C_VEL
LIN {X 0,Y 459.876,Z 506.377,A -85,B 0,C 180,E1 -8084.033,E2 -8084.033} C_VEL
LIN {X 0,Y 459.806,Z 510.748,A -85,B 0,C 180,E1 -8087.644,E2 -8087.644} C_VEL
LIN {X 0,Y 459.827,Z 511.142,A -85,B 0,C 180,E1 -8087.808,E2 -8087.808} C_VEL
LIN {X 0,Y 461.714,Z 521.667,A -85,B 0,C 180,E1 -8088.283,E2 -8088.283} C_VEL
LIN {X 0,Y 461.797,Z 529.583,A -85,B 0,C 180,E1 -8088.7,E2 -8088.7} C_VEL
LIN {X 0,Y 461.444,Z 539.471,A -85,B 0,C 180,E1 -8089.358,E2 -8089.358} C_VEL
LIN {X 0,Y 461.176,Z 547.362,A -85,B 0,C 180,E1 -8090.018,E2 -8090.018} C_VEL
LIN {X 0,Y 460.855,Z 554.93,A -85,B 0,C 180,E1 -8090.786,E2 -8090.786} C_VEL
LIN {X 0,Y 460.513,Z 563.674,A -85,B 0,C 180,E1 -8091.885,E2 -8091.885} C_VEL
LIN {X 0,Y 460.231,Z 570.644,A -85,B 0,C 180,E1 -8093.022,E2 -8093.022} C_VEL
LIN {X 0,Y 460.114,Z 574.896,A -85,B 0,C 180,E1 -8093.862,E2 -8093.862} C_VEL
LIN {X 0,Y 459.8,Z 578.62,A -85,B 0,C 180,E1 -8094.738,E2 -8094.738} C_VEL
LIN {X 0,Y 459.902,Z 581.623,A -85,B 0,C 180,E1 -8095.618,E2 -8095.618} C_VEL
LIN {X 0,Y 459.742,Z 583.97,A -85,B 0,C 180,E1 -8096.494,E2 -8096.494} C_VEL
LIN {X 0,Y 459.685,Z 585.758,A -85,B 0,C 180,E1 -8097.371,E2 -8097.371} C_VEL
LIN {X 0,Y 459.636,Z 587.038,A -85,B 0,C 180,E1 -8098.248,E2 -8098.248} C_VEL
LIN {X 0,Y 459.553,Z 587.836,A -85,B 0,C 180,E1 -8099.124,E2 -8099.124} C_VEL
LIN {X 0,Y 459.529,Z 588.114,A -85,B 0,C 180,E1 -8100,E2 -8100} C_VEL
LIN {X 0,Y 459.553,Z 587.8,A -85,B 0,C 180,E1 -8100.876,E2 -8100.876} C_VEL
LIN {X 0,Y 459.635,Z 587,A -85,B 0,C 180,E1 -8101.752,E2 -8101.752} C_VEL
LIN {X 0,Y 459.671,Z 585.719,A -85,B 0,C 180,E1 -8102.629,E2 -8102.629} C_VEL
LIN {X 0,Y 459.797,Z 582.75,A -85,B 0,C 180,E1 -8103.944,E2 -8103.944} C_VEL
LIN {X 0,Y 459.791,Z 580.055,A -85,B 0,C 180,E1 -8104.823,E2 -8104.823} C_VEL
LIN {X 0,Y 459.929,Z 576.726,A -85,B 0,C 180,E1 -8105.7,E2 -8105.7} C_VEL
LIN {X 0,Y 460.233,Z 572.122,A -85,B 0,C 180,E1 -8106.681,E2 -8106.681} C_VEL
LIN {X 0,Y 460.272,Z 566.397,A -85,B 0,C 180,E1 -8107.678,E2 -8107.678} C_VEL
LIN {X 0,Y 460.513,Z 560.243,A -85,B 0,C 180,E1 -8108.557,E2 -8108.557} C_VEL
LIN {X 0,Y 460.79,Z 553.797,A -85,B 0,C 180,E1 -8109.326,E2 -8109.326} C_VEL
LIN {X 0,Y 461.11,Z 546.028,A -85,B 0,C 180,E1 -8110.095,E2 -8110.095} C_VEL
LIN {X 0,Y 461.408,Z 537.885,A -85,B 0,C 180,E1 -8110.754,E2 -8110.754} C_VEL
LIN {X 0,Y 461.753,Z 527.648,A -85,B 0,C 180,E1 -8111.412,E2 -8111.412} C_VEL
LIN {X 0,Y 461.519,Z 520.116,A -85,B 0,C 180,E1 -8111.791,E2 -8111.791} C_VEL
LIN {X 0,Y 459.757,Z 509.425,A -85,B 0,C 180,E1 -8112.251,E2 -8112.251} C_VEL
LIN {X 0,Y 459.72,Z 504.139,A -85,B 0,C 180,E1 -8115.973,E2 -8115.973} C_VEL
LIN {X 0,Y 459.799,Z 500.293,A -85,B 0,C 180,E1 -8118.722,E2 -8118.722} C_VEL
LIN {X 0,Y 459.807,Z 496.442,A -85,B 0,C 180,E1 -8121.52,E2 -8121.52} C_VEL
LIN {X 0,Y 459.903,Z 492.565,A -85,B 0,C 180,E1 -8124.368,E2 -8124.368} C_VEL
LIN {X 0,Y 460.121,Z 489.023,A -85,B 0,C 180,E1 -8127.088,E2 -8127.088} C_VEL
LIN {X 0,Y 460.154,Z 494.573,A -85,B 0,C 180,E1 -8129.474,E2 -8129.474} C_VEL
LIN {X 0,Y 460.116,Z 502.268,A -85,B 0,C 180,E1 -8132.849,E2 -8132.849} C_VEL
LIN {X 0,Y 459.986,Z 509.24,A -85,B 0,C 180,E1 -8135.926,E2 -8135.926} C_VEL
LIN {X 0,Y 459.912,Z 516.92,A -85,B 0,C 180,E1 -8139.358,E2 -8139.358} C_VEL
LIN {X 0,Y 459.815,Z 524.546,A -85,B 0,C 180,E1 -8142.806,E2 -8142.806} C_VEL
LIN {X 0,Y 459.784,Z 526.645,A -85,B 0,C 180,E1 -8143.755,E2 -8143.755} C_VEL
LIN {X 0,Y 461.521,Z 537.559,A -85,B 0,C 180,E1 -8144.169,E2 -8144.169} C_VEL
LIN {X 0,Y 461.814,Z 543.084,A -85,B 0,C 180,E1 -8144.43,E2 -8144.43} C_VEL
LIN {X 0,Y 461.582,Z 551.973,A -85,B 0,C 180,E1 -8144.927,E2 -8144.927} C_VEL
LIN {X 0,Y 461.248,Z 561.163,A -85,B 0,C 180,E1 -8145.583,E2 -8145.583} C_VEL
LIN {X 0,Y 460.827,Z 571.233,A -85,B 0,C 180,E1 -8146.512,E2 -8146.512} C_VEL
LIN {X 0,Y 460.518,Z 579.126,A -85,B 0,C 180,E1 -8147.448,E2 -8147.448} C_VEL
LIN {X 0,Y 460.266,Z 584.177,A -85,B 0,C 180,E1 -8148.159,E2 -8148.159} C_VEL
LIN {X 0,Y 460.014,Z 590.13,A -85,B 0,C 180,E1 -8149.175,E2 -8149.175} C_VEL
LIN {X 0,Y 459.864,Z 594.433,A -85,B 0,C 180,E1 -8150.068,E2 -8150.068} C_VEL
LIN {X 0,Y 459.729,Z 598.889,A -85,B 0,C 180,E1 -8151.229,E2 -8151.229} C_VEL
LIN {X 0,Y 459.645,Z 602.009,A -85,B 0,C 180,E1 -8152.294,E2 -8152.294} C_VEL
LIN {X 0,Y 459.548,Z 604.332,A -85,B 0,C 180,E1 -8153.384,E2 -8153.384} C_VEL
LIN {X 0,Y 459.477,Z 605.821,A -85,B 0,C 180,E1 -8154.462,E2 -8154.462} C_VEL
LIN {X 0,Y 459.428,Z 606.598,A -85,B 0,C 180,E1 -8155.696,E2 -8155.696} C_VEL
LIN {X 0,Y 459.43,Z 606.171,A -85,B 0,C 180,E1 -8157.283,E2 -8157.283} C_VEL
LIN {X 0,Y 459.563,Z 603.913,A -85,B 0,C 180,E1 -8158.915,E2 -8158.915} C_VEL
LIN {X 0,Y 459.64,Z 600.923,A -85,B 0,C 180,E1 -8160.197,E2 -8160.197} C_VEL
LIN {X 0,Y 459.753,Z 597.621,A -85,B 0,C 180,E1 -8161.215,E2 -8161.215} C_VEL
LIN {X 0,Y 459.947,Z 592.652,A -85,B 0,C 180,E1 -8162.405,E2 -8162.405} C_VEL
LIN {X 0,Y 460.17,Z 586.95,A -85,B 0,C 180,E1 -8163.466,E2 -8163.466} C_VEL
LIN {X 0,Y 460.426,Z 580.203,A -85,B 0,C 180,E1 -8164.479,E2 -8164.479} C_VEL
LIN {X 0,Y 460.684,Z 573.42,A -85,B 0,C 180,E1 -8165.315,E2 -8165.315} C_VEL
LIN {X 0,Y 460.981,Z 567.141,A -85,B 0,C 180,E1 -8165.962,E2 -8165.962} C_VEL
LIN {X 0,Y 461.244,Z 558.959,A -85,B 0,C 180,E1 -8166.661,E2 -8166.661} C_VEL
LIN {X 0,Y 461.506,Z 553.236,A -85,B 0,C 180,E1 -8167.069,E2 -8167.069} C_VEL
LIN {X 0,Y 460.8,Z 549.226,A -85,B 0,C 180,E1 -8167.342,E2 -8167.342} C_VEL
LIN {X 0,Y 458.136,Z 544.464,A -85,B 0,C 180,E1 -8167.671,E2 -8167.671} C_VEL
LIN {X 0,Y 455.09,Z 539.056,A -85,B 0,C 180,E1 -8168.02,E2 -8168.02} C_VEL
LIN {X 0,Y 454.003,Z 535.425,A -85,B 0,C 180,E1 -8168.189,E2 -8168.189} C_VEL
LIN {X 0,Y 452.6,Z 526.938,A -85,B 0,C 180,E1 -8168.508,E2 -8168.508} C_VEL
LIN {X 0,Y 452.7,Z 519.964,A -85,B 0,C 180,E1 -8171.911,E2 -8171.911} C_VEL
LIN {X 0,Y 452.778,Z 514.238,A -85,B 0,C 180,E1 -8174.7,E2 -8174.7} C_VEL
LIN {X 0,Y 452.954,Z 506.726,A -85,B 0,C 180,E1 -8178.363,E2 -8178.363} C_VEL
LIN {X 0,Y 453.009,Z 501.164,A -85,B 0,C 180,E1 -8181.075,E2 -8181.075} C_VEL
LIN {X 0,Y 453.075,Z 495.578,A -85,B 0,C 180,E1 -8183.766,E2 -8183.766} C_VEL
LIN {X 0,Y 453.244,Z 491.793,A -85,B 0,C 180,E1 -8185.553,E2 -8185.553} C_VEL
LIN {X 0,Y 453.129,Z 488.858,A -85,B 0,C 180,E1 -8186.999,E2 -8186.999} C_VEL
LIN {X 0,Y 453.65,Z 488.79,A -85,B 0,C 180,E1 -8189.112,E2 -8189.112} C_VEL
LIN {X 0,Y 453.718,Z 488.781,A -85,B 0,C 180,E1 -8190.887,E2 -8190.887} C_VEL
LIN {X 0,Y 453.766,Z 488.777,A -85,B 0,C 180,E1 -8192.663,E2 -8192.663} C_VEL
LIN {X 0,Y 453.68,Z 488.787,A -85,B 0,C 180,E1 -8196.225,E2 -8196.225} C_VEL
LIN {X 0,Y 453.592,Z 488.797,A -85,B 0,C 180,E1 -8198.913,E2 -8198.913} C_VEL
LIN {X 0,Y 453.564,Z 488.801,A -85,B 0,C 180,E1 -8202.528,E2 -8202.528} C_VEL
LIN {X 0,Y 453.545,Z 488.804,A -85,B 0,C 180,E1 -8206.195,E2 -8206.195} C_VEL
LIN {X 0,Y 453.521,Z 488.805,A -85,B 0,C 180,E1 -8209.04,E2 -8209.04} C_VEL
LIN {X 0,Y 453.477,Z 488.812,A -85,B 0,C 180,E1 -8211.836,E2 -8211.836} C_VEL
LIN {X 0,Y 453.515,Z 488.807,A -85,B 0,C 180,E1 -8214.734,E2 -8214.734} C_VEL
LIN {X 0,Y 453.539,Z 488.806,A -85,B 0,C 180,E1 -8217.961,E2 -8217.961} C_VEL
LIN {X 0,Y 453.483,Z 488.811,A -85,B 0,C 180,E1 -8220.758,E2 -8220.758} C_VEL
LIN {X 0,Y 453.477,Z 488.813,A -85,B 0,C 180,E1 -8223.912,E2 -8223.912} C_VEL
LIN {X 0,Y 453.47,Z 488.812,A -85,B 0,C 180,E1 -8227.187,E2 -8227.187} C_VEL
LIN {X 0,Y 453.516,Z 488.806,A -85,B 0,C 180,E1 -8229.446,E2 -8229.446} C_VEL
LIN {X 0,Y 453.466,Z 488.812,A -85,B 0,C 180,E1 -8232.994,E2 -8232.994} C_VEL
LIN {X 0,Y 453.475,Z 488.813,A -85,B 0,C 180,E1 -8235.78,E2 -8235.78} C_VEL
LIN {X 0,Y 453.495,Z 488.81,A -85,B 0,C 180,E1 -8238.211,E2 -8238.211} C_VEL
LIN {X 0,Y 453.529,Z 488.804,A -85,B 0,C 180,E1 -8240.787,E2 -8240.787} C_VEL
LIN {X 0,Y 453.452,Z 488.816,A -85,B 0,C 180,E1 -8243.917,E2 -8243.917} C_VEL
LIN {X 0,Y 453.481,Z 488.81,A -85,B 0,C 180,E1 -8247.151,E2 -8247.151} C_VEL
LIN {X 0,Y 453.473,Z 488.813,A -85,B 0,C 180,E1 -8250.268,E2 -8250.268} C_VEL
LIN {X 0,Y 453.512,Z 488.807,A -85,B 0,C 180,E1 -8253.294,E2 -8253.294} C_VEL
LIN {X 0,Y 453.502,Z 488.809,A -85,B 0,C 180,E1 -8256.239,E2 -8256.239} C_VEL
LIN {X 0,Y 453.481,Z 488.811,A -85,B 0,C 180,E1 -8259.117,E2 -8259.117} C_VEL
LIN {X 0,Y 453.51,Z 488.808,A -85,B 0,C 180,E1 -8261.944,E2 -8261.944} C_VEL
LIN {X 0,Y 453.537,Z 488.803,A -85,B 0,C 180,E1 -8264.726,E2 -8264.726} C_VEL
LIN {X 0,Y 453.6,Z 488.798,A -85,B 0,C 180,E1 -8267.472,E2 -8267.472} C_VEL
LIN {X 0,Y 453.59,Z 488.797,A -85,B 0,C 180,E1 -8271.087,E2 -8271.087} C_VEL
LIN {X 0,Y 453.675,Z 488.788,A -85,B 0,C 180,E1 -8273.775,E2 -8273.775} C_VEL
LIN {X 0,Y 453.764,Z 488.776,A -85,B 0,C 180,E1 -8277.337,E2 -8277.337} C_VEL
LIN {X 0,Y 453.821,Z 488.77,A -85,B 0,C 180,E1 -8280,E2 -8280} C_VEL
LIN {X 0,Y 453.764,Z 488.775,A -85,B 0,C 180,E1 -8282.663,E2 -8282.663} C_VEL
LIN {X 0,Y 453.676,Z 488.787,A -85,B 0,C 180,E1 -8286.225,E2 -8286.225} C_VEL
LIN {X 0,Y 453.59,Z 488.797,A -85,B 0,C 180,E1 -8288.913,E2 -8288.913} C_VEL
LIN {X 0,Y 453.56,Z 488.799,A -85,B 0,C 180,E1 -8292.529,E2 -8292.529} C_VEL
LIN {X 0,Y 453.542,Z 488.803,A -85,B 0,C 180,E1 -8296.196,E2 -8296.196} C_VEL
LIN {X 0,Y 453.518,Z 488.805,A -85,B 0,C 180,E1 -8299.041,E2 -8299.041} C_VEL
LIN {X 0,Y 453.474,Z 488.813,A -85,B 0,C 180,E1 -8301.836,E2 -8301.836} C_VEL
LIN {X 0,Y 453.511,Z 488.805,A -85,B 0,C 180,E1 -8304.734,E2 -8304.734} C_VEL
LIN {X 0,Y 453.536,Z 488.804,A -85,B 0,C 180,E1 -8307.961,E2 -8307.961} C_VEL
LIN {X 0,Y 453.481,Z 488.81,A -85,B 0,C 180,E1 -8310.759,E2 -8310.759} C_VEL
LIN {X 0,Y 453.475,Z 488.812,A -85,B 0,C 180,E1 -8313.913,E2 -8313.913} C_VEL
LIN {X 0,Y 453.468,Z 488.815,A -85,B 0,C 180,E1 -8317.188,E2 -8317.188} C_VEL
LIN {X 0,Y 453.502,Z 488.81,A -85,B 0,C 180,E1 -8319.448,E2 -8319.448} C_VEL
LIN {X 0,Y 453.466,Z 488.814,A -85,B 0,C 180,E1 -8322.995,E2 -8322.995} C_VEL
LIN {X 0,Y 453.464,Z 488.814,A -85,B 0,C 180,E1 -8325.779,E2 -8325.779} C_VEL
LIN {X 0,Y 453.514,Z 488.808,A -85,B 0,C 180,E1 -8329.406,E2 -8329.406} C_VEL
LIN {X 0,Y 453.476,Z 488.813,A -85,B 0,C 180,E1 -8332.223,E2 -8332.223} C_VEL
LIN {X 0,Y 453.554,Z 488.944,A -85,B 0,C 180,E1 -8335.018,E2 -8335.018} C_VEL
LIN {X 0,Y 454.827,Z 496.647,A -85,B 0,C 180,E1 -8338.196,E2 -8338.196} C_VEL
LIN {X 0,Y 454.638,Z 502.221,A -85,B 0,C 180,E1 -8340.353,E2 -8340.353} C_VEL
LIN {X 0,Y 454.17,Z 510.158,A -85,B 0,C 180,E1 -8343.337,E2 -8343.337} C_VEL
LIN {X 0,Y 453.786,Z 518.109,A -85,B 0,C 180,E1 -8346.255,E2 -8346.255} C_VEL
LIN {X 0,Y 453.395,Z 527.388,A -85,B 0,C 180,E1 -8349.588,E2 -8349.588} C_VEL
LIN {X 0,Y 453.045,Z 536.685,A -85,B 0,C 180,E1 -8352.858,E2 -8352.858} C_VEL
LIN {X 0,Y 452.819,Z 545.971,A -85,B 0,C 180,E1 -8356.08,E2 -8356.08} C_VEL
LIN {X 0,Y 452.773,Z 550.339,A -85,B 0,C 180,E1 -8357.547,E2 -8357.547} C_VEL
LIN {X 0,Y 454.014,Z 562.132,A -85,B 0,C 180,E1 -8357.978,E2 -8357.978} C_VEL
LIN {X 0,Y 454.48,Z 570.612,A -85,B 0,C 180,E1 -8358.403,E2 -8358.403} C_VEL
LIN {X 0,Y 454.173,Z 581.04,A -85,B 0,C 180,E1 -8359.073,E2 -8359.073} C_VEL
LIN {X 0,Y 453.801,Z 589.284,A -85,B 0,C 180,E1 -8359.741,E2 -8359.741} C_VEL
LIN {X 0,Y 453.452,Z 597.139,A -85,B 0,C 180,E1 -8360.522,E2 -8360.522} C_VEL
LIN {X 0,Y 453.212,Z 603.665,A -85,B 0,C 180,E1 -8361.304,E2 -8361.304} C_VEL
LIN {X 0,Y 452.954,Z 609.889,A -85,B 0,C 180,E1 -8362.198,E2 -8362.198} C_VEL
LIN {X 0,Y 452.831,Z 615.067,A -85,B 0,C 180,E1 -8363.092,E2 -8363.092} C_VEL
LIN {X 0,Y 452.672,Z 620.338,A -85,B 0,C 180,E1 -8364.209,E2 -8364.209} C_VEL
LIN {X 0,Y 452.526,Z 625.23,A -85,B 0,C 180,E1 -8365.547,E2 -8365.547} C_VEL
LIN {X 0,Y 452.556,Z 627.611,A -85,B 0,C 180,E1 -8366.439,E2 -8366.439} C_VEL
LIN {X 0,Y 452.533,Z 629.423,A -85,B 0,C 180,E1 -8367.33,E2 -8367.33} C_VEL
LIN {X 0,Y 452.482,Z 630.717,A -85,B 0,C 180,E1 -8368.22,E2 -8368.22} C_VEL
LIN {X 0,Y 452.486,Z 631.518,A -85,B 0,C 180,E1 -8369.111,E2 -8369.111} C_VEL
LIN {X 0,Y 452.461,Z 631.796,A -85,B 0,C 180,E1 -8370,E2 -8370} C_VEL
LIN {X 0,Y 452.486,Z 631.473,A -85,B 0,C 180,E1 -8370.89,E2 -8370.89} C_VEL
LIN {X 0,Y 452.483,Z 630.651,A -85,B 0,C 180,E1 -8371.781,E2 -8371.781} C_VEL
LIN {X 0,Y 452.534,Z 629.335,A -85,B 0,C 180,E1 -8372.671,E2 -8372.671} C_VEL
LIN {X 0,Y 452.526,Z 626.294,A -85,B 0,C 180,E1 -8374.008,E2 -8374.008} C_VEL
LIN {X 0,Y 452.592,Z 623.536,A -85,B 0,C 180,E1 -8374.9,E2 -8374.9} C_VEL
LIN {X 0,Y 452.709,Z 618.176,A -85,B 0,C 180,E1 -8376.239,E2 -8376.239} C_VEL
LIN {X 0,Y 452.903,Z 611.094,A -85,B 0,C 180,E1 -8377.58,E2 -8377.58} C_VEL
LIN {X 0,Y 453.196,Z 603.431,A -85,B 0,C 180,E1 -8378.697,E2 -8378.697} C_VEL
LIN {X 0,Y 453.524,Z 595.902,A -85,B 0,C 180,E1 -8379.59,E2 -8379.59} C_VEL
LIN {X 0,Y 453.863,Z 587.885,A -85,B 0,C 180,E1 -8380.371,E2 -8380.371} C_VEL
LIN {X 0,Y 454.255,Z 577.974,A -85,B 0,C 180,E1 -8381.151,E2 -8381.151} C_VEL
LIN {X 0,Y 454.433,Z 567.598,A -85,B 0,C 180,E1 -8381.77,E2 -8381.77} C_VEL
LIN {X 0,Y 453.57,Z 557.599,A -85,B 0,C 180,E1 -8382.245,E2 -8382.245} C_VEL
LIN {X 0,Y 452.675,Z 549.296,A -85,B 0,C 180,E1 -8382.554,E2 -8382.554} C_VEL
LIN {X 0,Y 452.858,Z 540.262,A -85,B 0,C 180,E1 -8385.806,E2 -8385.806} C_VEL
LIN {X 0,Y 453.074,Z 531.588,A -85,B 0,C 180,E1 -8389.011,E2 -8389.011} C_VEL
LIN {X 0,Y 453.316,Z 524.167,A -85,B 0,C 180,E1 -8391.845,E2 -8391.845} C_VEL
LIN {X 0,Y 453.644,Z 516.962,A -85,B 0,C 180,E1 -8394.727,E2 -8394.727} C_VEL
LIN {X 0,Y 454.138,Z 509.043,A -85,B 0,C 180,E1 -8398.103,E2 -8398.103} C_VEL
LIN {X 0,Y 454.732,Z 502.479,A -85,B 0,C 180,E1 -8401.182,E2 -8401.182} C_VEL
LIN {X 0,Y 454.933,Z 498.141,A -85,B 0,C 180,E1 -8403.466,E2 -8403.466} C_VEL
LIN {X 0,Y 454.418,Z 494.132,A -85,B 0,C 180,E1 -8405.995,E2 -8405.995} C_VEL
LIN {X 0,Y 453.881,Z 491.175,A -85,B 0,C 180,E1 -8408.271,E2 -8408.271} C_VEL
LIN {X 0,Y 453.496,Z 488.811,A -85,B 0,C 180,E1 -8410.609,E2 -8410.609} C_VEL
LIN {X 0,Y 453.458,Z 488.816,A -85,B 0,C 180,E1 -8413.245,E2 -8413.245} C_VEL
LIN {X 0,Y 453.476,Z 488.812,A -85,B 0,C 180,E1 -8415.78,E2 -8415.78} C_VEL
LIN {X 0,Y 453.484,Z 488.812,A -85,B 0,C 180,E1 -8418.21,E2 -8418.21} C_VEL
LIN {X 0,Y 453.512,Z 488.809,A -85,B 0,C 180,E1 -8420.791,E2 -8420.791} C_VEL
LIN {X 0,Y 453.456,Z 488.816,A -85,B 0,C 180,E1 -8423.917,E2 -8423.917} C_VEL
LIN {X 0,Y 453.484,Z 488.813,A -85,B 0,C 180,E1 -8425.224,E2 -8425.224} C_VEL
LIN {X 0,Y 453.605,Z 490.095,A -85,B 0,C 180,E1 -8427.161,E2 -8427.161} C_VEL
LIN {X 0,Y 453.517,Z 492.678,A -85,B 0,C 180,E1 -8430.271,E2 -8430.271} C_VEL
LIN {X 0,Y 453.263,Z 495.504,A -85,B 0,C 180,E1 -8433.279,E2 -8433.279} C_VEL
LIN {X 0,Y 453.094,Z 498.492,A -85,B 0,C 180,E1 -8436.229,E2 -8436.229} C_VEL
LIN {X 0,Y 452.977,Z 501.555,A -85,B 0,C 180,E1 -8439.093,E2 -8439.093} C_VEL
LIN {X 0,Y 452.862,Z 504.709,A -85,B 0,C 180,E1 -8441.918,E2 -8441.918} C_VEL
LIN {X 0,Y 452.837,Z 507.925,A -85,B 0,C 180,E1 -8444.702,E2 -8444.702} C_VEL
LIN {X 0,Y 452.77,Z 511.557,A -85,B 0,C 180,E1 -8447.586,E2 -8447.586} C_VEL
LIN {X 0,Y 454.667,Z 521.495,A -85,B 0,C 180,E1 -8448.052,E2 -8448.052} C_VEL
LIN {X 0,Y 454.953,Z 526.423,A -85,B 0,C 180,E1 -8448.311,E2 -8448.311} C_VEL
LIN {X 0,Y 454.633,Z 537.117,A -85,B 0,C 180,E1 -8448.971,E2 -8448.971} C_VEL
LIN {X 0,Y 454.245,Z 546.68,A -85,B 0,C 180,E1 -8449.751,E2 -8449.751} C_VEL
LIN {X 0,Y 453.914,Z 554.418,A -85,B 0,C 180,E1 -8450.531,E2 -8450.531} C_VEL
LIN {X 0,Y 453.64,Z 560.838,A -85,B 0,C 180,E1 -8451.312,E2 -8451.312} C_VEL
LIN {X 0,Y 453.351,Z 566.96,A -85,B 0,C 180,E1 -8452.204,E2 -8452.204} C_VEL
LIN {X 0,Y 453.204,Z 572.93,A -85,B 0,C 180,E1 -8453.269,E2 -8453.269} C_VEL
LIN {X 0,Y 452.749,Z 579.043,A -85,B 0,C 180,E1 -8454.656,E2 -8454.656} C_VEL
LIN {X 0,Y 452.845,Z 582.03,A -85,B 0,C 180,E1 -8455.55,E2 -8455.55} C_VEL
LIN {X 0,Y 452.685,Z 584.363,A -85,B 0,C 180,E1 -8456.44,E2 -8456.44} C_VEL
LIN {X 0,Y 452.607,Z 586.137,A -85,B 0,C 180,E1 -8457.33,E2 -8457.33} C_VEL
LIN {X 0,Y 452.576,Z 587.403,A -85,B 0,C 180,E1 -8458.22,E2 -8458.22} C_VEL
LIN {X 0,Y 452.489,Z 588.188,A -85,B 0,C 180,E1 -8459.11,E2 -8459.11} C_VEL
LIN {X 0,Y 452.463,Z 588.459,A -85,B 0,C 180,E1 -8460,E2 -8460} C_VEL
LIN {X 0,Y 452.489,Z 588.135,A -85,B 0,C 180,E1 -8460.89,E2 -8460.89} C_VEL
LIN {X 0,Y 452.545,Z 587.322,A -85,B 0,C 180,E1 -8461.78,E2 -8461.78} C_VEL
LIN {X 0,Y 452.593,Z 586.025,A -85,B 0,C 180,E1 -8462.67,E2 -8462.67} C_VEL
LIN {X 0,Y 452.739,Z 583.037,A -85,B 0,C 180,E1 -8464.006,E2 -8464.006} C_VEL
LIN {X 0,Y 452.706,Z 580.323,A -85,B 0,C 180,E1 -8464.898,E2 -8464.898} C_VEL
LIN {X 0,Y 452.893,Z 576.974,A -85,B 0,C 180,E1 -8465.789,E2 -8465.789} C_VEL
LIN {X 0,Y 453.162,Z 572.745,A -85,B 0,C 180,E1 -8466.711,E2 -8466.711} C_VEL
LIN {X 0,Y 453.228,Z 566.593,A -85,B 0,C 180,E1 -8467.798,E2 -8467.798} C_VEL
LIN {X 0,Y 453.498,Z 560.41,A -85,B 0,C 180,E1 -8468.691,E2 -8468.691} C_VEL
LIN {X 0,Y 453.798,Z 553.935,A -85,B 0,C 180,E1 -8469.471,E2 -8469.471} C_VEL
LIN {X 0,Y 454.133,Z 546.134,A -85,B 0,C 180,E1 -8470.252,E2 -8470.252} C_VEL
LIN {X 0,Y 454.436,Z 537.956,A -85,B 0,C 180,E1 -8470.921,E2 -8470.921} C_VEL
LIN {X 0,Y 454.786,Z 527.672,A -85,B 0,C 180,E1 -8471.589,E2 -8471.589} C_VEL
LIN {X 0,Y 454.588,Z 521.256,A -85,B 0,C 180,E1 -8471.917,E2 -8471.917} C_VEL
LIN {X 0,Y 452.677,Z 509.702,A -85,B 0,C 180,E1 -8472.431,E2 -8472.431} C_VEL
LIN {X 0,Y 452.681,Z 505.056,A -85,B 0,C 180,E1 -8475.725,E2 -8475.725} C_VEL
LIN {X 0,Y 452.726,Z 500.478,A -85,B 0,C 180,E1 -8479.026,E2 -8479.026} C_VEL
LIN {X 0,Y 452.729,Z 496.593,A -85,B 0,C 180,E1 -8481.874,E2 -8481.874} C_VEL
LIN {X 0,Y 452.876,Z 492.689,A -85,B 0,C 180,E1 -8484.772,E2 -8484.772} C_VEL
LIN {X 0,Y 453.069,Z 489.818,A -85,B 0,C 180,E1 -8487.045,E2 -8487.045} C_VEL
LIN {X 0,Y 453.109,Z 496.028,A -85,B 0,C 180,E1 -8489.758,E2 -8489.758} C_VEL
LIN {X 0,Y 453.052,Z 503.598,A -85,B 0,C 180,E1 -8493.103,E2 -8493.103} C_VEL
LIN {X 0,Y 452.904,Z 510.557,A -85,B 0,C 180,E1 -8496.203,E2 -8496.203} C_VEL
LIN {X 0,Y 452.838,Z 517.011,A -85,B 0,C 180,E1 -8499.104,E2 -8499.104} C_VEL
LIN {X 0,Y 452.732,Z 524.435,A -85,B 0,C 180,E1 -8502.475,E2 -8502.475} C_VEL
LIN {X 0,Y 452.734,Z 526.804,A -85,B 0,C 180,E1 -8503.556,E2 -8503.556} C_VEL
LIN {X 0,Y 454.525,Z 537.878,A -85,B 0,C 180,E1 -8503.985,E2 -8503.985} C_VEL
LIN {X 0,Y 454.892,Z 542.683,A -85,B 0,C 180,E1 -8504.218,E2 -8504.218} C_VEL
LIN {X 0,Y 454.69,Z 551.056,A -85,B 0,C 180,E1 -8504.682,E2 -8504.682} C_VEL
LIN {X 0,Y 454.339,Z 559.211,A -85,B 0,C 180,E1 -8505.25,E2 -8505.25} C_VEL
LIN {X 0,Y 454.018,Z 567.504,A -85,B 0,C 180,E1 -8505.971,E2 -8505.971} C_VEL
LIN {X 0,Y 453.645,Z 575.899,A -85,B 0,C 180,E1 -8506.871,E2 -8506.871} C_VEL
LIN {X 0,Y 453.288,Z 583.432,A -85,B 0,C 180,E1 -8507.884,E2 -8507.884} C_VEL
LIN {X 0,Y 452.959,Z 590.181,A -85,B 0,C 180,E1 -8509.039,E2 -8509.039} C_VEL
LIN {X 0,Y 452.778,Z 595.688,A -85,B 0,C 180,E1 -8510.229,E2 -8510.229} C_VEL
LIN {X 0,Y 452.621,Z 600.565,A -85,B 0,C 180,E1 -8511.603,E2 -8511.603} C_VEL
LIN {X 0,Y 452.535,Z 603.403,A -85,B 0,C 180,E1 -8512.722,E2 -8512.722} C_VEL
LIN {X 0,Y 452.439,Z 605.418,A -85,B 0,C 180,E1 -8513.876,E2 -8513.876} C_VEL
LIN {X 0,Y 452.349,Z 606.491,A -85,B 0,C 180,E1 -8514.91,E2 -8514.91} C_VEL
LIN {X 0,Y 452.317,Z 606.883,A -85,B 0,C 180,E1 -8515.988,E2 -8515.988} C_VEL
LIN {X 0,Y 452.332,Z 606.544,A -85,B 0,C 180,E1 -8517.057,E2 -8517.057} C_VEL
LIN {X 0,Y 452.398,Z 605.49,A -85,B 0,C 180,E1 -8518.116,E2 -8518.116} C_VEL
LIN {X 0,Y 452.523,Z 602.563,A -85,B 0,C 180,E1 -8519.685,E2 -8519.685} C_VEL
LIN {X 0,Y 452.621,Z 599.371,A -85,B 0,C 180,E1 -8520.822,E2 -8520.822} C_VEL
LIN {X 0,Y 452.811,Z 593.949,A -85,B 0,C 180,E1 -8522.249,E2 -8522.249} C_VEL
LIN {X 0,Y 453.115,Z 587.692,A -85,B 0,C 180,E1 -8523.487,E2 -8523.487} C_VEL
LIN {X 0,Y 453.382,Z 581.011,A -85,B 0,C 180,E1 -8524.522,E2 -8524.522} C_VEL
LIN {X 0,Y 453.686,Z 573.455,A -85,B 0,C 180,E1 -8525.472,E2 -8525.472} C_VEL
LIN {X 0,Y 454.052,Z 565.661,A -85,B 0,C 180,E1 -8526.269,E2 -8526.269} C_VEL
LIN {X 0,Y 454.377,Z 556.712,A -85,B 0,C 180,E1 -8527.011,E2 -8527.011} C_VEL
LIN {X 0,Y 454.77,Z 545.832,A -85,B 0,C 180,E1 -8527.691,E2 -8527.691} C_VEL
LIN {X 0,Y 454.665,Z 540.101,A -85,B 0,C 180,E1 -8527.985,E2 -8527.985} C_VEL
LIN {X 0,Y 454.003,Z 535.425,A -85,B 0,C 180,E1 -8528.189,E2 -8528.189} C_VEL
LIN {X 0,Y 453.241,Z 532.133,A -85,B 0,C 180,E1 -8528.406,E2 -8528.406} C_VEL
LIN {X 0,Y 451.729,Z 528.879,A -85,B 0,C 180,E1 -8528.81,E2 -8528.81} C_VEL
LIN {X 0,Y 449.967,Z 526.471,A -85,B 0,C 180,E1 -8529.305,E2 -8529.305} C_VEL
LIN {X 0,Y 447.866,Z 524.418,A -85,B 0,C 180,E1 -8529.995,E2 -8529.995} C_VEL
LIN {X 0,Y 445.876,Z 522.375,A -85,B 0,C 180,E1 -8531.002,E2 -8531.002} C_VEL
LIN {X 0,Y 445.593,Z 521.345,A -85,B 0,C 180,E1 -8531.522,E2 -8531.522} C_VEL
LIN {X 0,Y 445.699,Z 515.375,A -85,B 0,C 180,E1 -8534.45,E2 -8534.45} C_VEL
LIN {X 0,Y 445.887,Z 507.791,A -85,B 0,C 180,E1 -8538.176,E2 -8538.176} C_VEL
LIN {X 0,Y 445.941,Z 502.177,A -85,B 0,C 180,E1 -8540.932,E2 -8540.932} C_VEL
LIN {X 0,Y 446.022,Z 496.534,A -85,B 0,C 180,E1 -8543.667,E2 -8543.667} C_VEL
LIN {X 0,Y 446.184,Z 492.738,A -85,B 0,C 180,E1 -8545.482,E2 -8545.482} C_VEL
LIN {X 0,Y 446.094,Z 489.734,A -85,B 0,C 180,E1 -8546.952,E2 -8546.952} C_VEL
LIN {X 0,Y 446.607,Z 489.667,A -85,B 0,C 180,E1 -8549.098,E2 -8549.098} C_VEL
LIN {X 0,Y 446.789,Z 489.645,A -85,B 0,C 180,E1 -8550,E2 -8550} C_VEL
LIN {X 0,Y 446.71,Z 489.656,A -85,B 0,C 180,E1 -8552.705,E2 -8552.705} C_VEL
LIN {X 0,Y 446.649,Z 489.664,A -85,B 0,C 180,E1 -8556.323,E2 -8556.323} C_VEL
LIN {X 0,Y 446.538,Z 489.674,A -85,B 0,C 180,E1 -8559.055,E2 -8559.055} C_VEL
LIN {X 0,Y 446.522,Z 489.678,A -85,B 0,C 180,E1 -8562.729,E2 -8562.729} C_VEL
LIN {X 0,Y 446.497,Z 489.682,A -85,B 0,C 180,E1 -8566.227,E2 -8566.227} C_VEL
LIN {X 0,Y 446.47,Z 489.683,A -85,B 0,C 180,E1 -8569.303,E2 -8569.303} C_VEL
LIN {X 0,Y 446.419,Z 489.692,A -85,B 0,C 180,E1 -8572.199,E2 -8572.199} C_VEL
LIN {X 0,Y 446.459,Z 489.685,A -85,B 0,C 180,E1 -8575.152,E2 -8575.152} C_VEL
LIN {X 0,Y 446.484,Z 489.684,A -85,B 0,C 180,E1 -8578.178,E2 -8578.178} C_VEL
LIN {X 0,Y 446.419,Z 489.69,A -85,B 0,C 180,E1 -8581.299,E2 -8581.299} C_VEL
LIN {X 0,Y 446.43,Z 489.691,A -85,B 0,C 180,E1 -8584.522,E2 -8584.522} C_VEL
LIN {X 0,Y 446.43,Z 489.691,A -85,B 0,C 180,E1 -8588.081,E2 -8588.081} C_VEL
LIN {X 0,Y 446.426,Z 489.688,A -85,B 0,C 180,E1 -8590.917,E2 -8590.917} C_VEL
LIN {X 0,Y 446.421,Z 489.691,A -85,B 0,C 180,E1 -8593.843,E2 -8593.843} C_VEL
LIN {X 0,Y 446.445,Z 489.689,A -85,B 0,C 180,E1 -8596.396,E2 -8596.396} C_VEL
LIN {X 0,Y 446.467,Z 489.685,A -85,B 0,C 180,E1 -8599.805,E2 -8599.805} C_VEL
LIN {X 0,Y 446.431,Z 489.69,A -85,B 0,C 180,E1 -8602.123,E2 -8602.123} C_VEL
LIN {X 0,Y 446.426,Z 489.69,A -85,B 0,C 180,E1 -8605.477,E2 -8605.477} C_VEL
LIN {X 0,Y 446.414,Z 489.69,A -85,B 0,C 180,E1 -8608.699,E2 -8608.699} C_VEL
LIN {X 0,Y 446.482,Z 489.684,A -85,B 0,C 180,E1 -8611.821,E2 -8611.821} C_VEL
LIN {X 0,Y 446.456,Z 489.684,A -85,B 0,C 180,E1 -8614.848,E2 -8614.848} C_VEL
LIN {X 0,Y 446.446,Z 489.688,A -85,B 0,C 180,E1 -8618.245,E2 -8618.245} C_VEL
LIN {X 0,Y 446.456,Z 489.688,A -85,B 0,C 180,E1 -8621.649,E2 -8621.649} C_VEL
LIN {X 0,Y 446.505,Z 489.68,A -85,B 0,C 180,E1 -8624.48,E2 -8624.48} C_VEL
LIN {X 0,Y 446.537,Z 489.677,A -85,B 0,C 180,E1 -8628.194,E2 -8628.194} C_VEL
LIN {X 0,Y 446.598,Z 489.67,A -85,B 0,C 180,E1 -8631.858,E2 -8631.858} C_VEL
LIN {X 0,Y 446.643,Z 489.662,A -85,B 0,C 180,E1 -8634.583,E2 -8634.583} C_VEL
LIN {X 0,Y 446.708,Z 489.655,A -85,B 0,C 180,E1 -8637.295,E2 -8637.295} C_VEL
LIN {X 0,Y 446.792,Z 489.646,A -85,B 0,C 180,E1 -8640,E2 -8640} C_VEL
LIN {X 0,Y 446.708,Z 489.654,A -85,B 0,C 180,E1 -8642.705,E2 -8642.705} C_VEL
LIN {X 0,Y 446.645,Z 489.662,A -85,B 0,C 180,E1 -8646.324,E2 -8646.324} C_VEL
LIN {X 0,Y 446.536,Z 489.676,A -85,B 0,C 180,E1 -8649.055,E2 -8649.055} C_VEL
LIN {X 0,Y 446.518,Z 489.676,A -85,B 0,C 180,E1 -8652.73,E2 -8652.73} C_VEL
LIN {X 0,Y 446.493,Z 489.681,A -85,B 0,C 180,E1 -8656.228,E2 -8656.228} C_VEL
LIN {X 0,Y 446.467,Z 489.686,A -85,B 0,C 180,E1 -8659.303,E2 -8659.303} C_VEL
LIN {X 0,Y 446.416,Z 489.691,A -85,B 0,C 180,E1 -8662.2,E2 -8662.2} C_VEL
LIN {X 0,Y 446.455,Z 489.686,A -85,B 0,C 180,E1 -8665.152,E2 -8665.152} C_VEL
LIN {X 0,Y 446.481,Z 489.683,A -85,B 0,C 180,E1 -8668.179,E2 -8668.179} C_VEL
LIN {X 0,Y 446.418,Z 489.693,A -85,B 0,C 180,E1 -8671.3,E2 -8671.3} C_VEL
LIN {X 0,Y 446.428,Z 489.689,A -85,B 0,C 180,E1 -8674.523,E2 -8674.523} C_VEL
LIN {X 0,Y 446.428,Z 489.69,A -85,B 0,C 180,E1 -8678.082,E2 -8678.082} C_VEL
LIN {X 0,Y 446.425,Z 489.69,A -85,B 0,C 180,E1 -8680.918,E2 -8680.918} C_VEL
LIN {X 0,Y 446.42,Z 489.692,A -85,B 0,C 180,E1 -8683.843,E2 -8683.843} C_VEL
LIN {X 0,Y 446.397,Z 489.693,A -85,B 0,C 180,E1 -8686.404,E2 -8686.404} C_VEL
LIN {X 0,Y 446.467,Z 489.686,A -85,B 0,C 180,E1 -8689.805,E2 -8689.805} C_VEL
LIN {X 0,Y 446.433,Z 489.69,A -85,B 0,C 180,E1 -8692.124,E2 -8692.124} C_VEL
LIN {X 0,Y 446.489,Z 489.69,A -85,B 0,C 180,E1 -8694.778,E2 -8694.778} C_VEL
LIN {X 0,Y 447.759,Z 497.224,A -85,B 0,C 180,E1 -8697.949,E2 -8697.949} C_VEL
LIN {X 0,Y 447.717,Z 502.016,A -85,B 0,C 180,E1 -8699.847,E2 -8699.847} C_VEL
LIN {X 0,Y 447.213,Z 509.942,A -85,B 0,C 180,E1 -8702.888,E2 -8702.888} C_VEL
LIN {X 0,Y 446.785,Z 517.875,A -85,B 0,C 180,E1 -8705.86,E2 -8705.86} C_VEL
LIN {X 0,Y 446.384,Z 527.135,A -85,B 0,C 180,E1 -8709.253,E2 -8709.253} C_VEL
LIN {X 0,Y 446.012,Z 536.411,A -85,B 0,C 180,E1 -8712.579,E2 -8712.579} C_VEL
LIN {X 0,Y 445.752,Z 545.662,A -85,B 0,C 180,E1 -8715.855,E2 -8715.855} C_VEL
LIN {X 0,Y 445.69,Z 549.964,A -85,B 0,C 180,E1 -8717.359,E2 -8717.359} C_VEL
LIN {X 0,Y 447.011,Z 562.818,A -85,B 0,C 180,E1 -8717.855,E2 -8717.855} C_VEL
LIN {X 0,Y 447.51,Z 569.919,A -85,B 0,C 180,E1 -8718.22,E2 -8718.22} C_VEL
LIN {X 0,Y 447.136,Z 580.439,A -85,B 0,C 180,E1 -8718.899,E2 -8718.899} C_VEL
LIN {X 0,Y 446.762,Z 588.738,A -85,B 0,C 180,E1 -8719.578,E2 -8719.578} C_VEL
LIN {X 0,Y 446.438,Z 596.635,A -85,B 0,C 180,E1 -8720.372,E2 -8720.372} C_VEL
LIN {X 0,Y 446.157,Z 603.192,A -85,B 0,C 180,E1 -8721.166,E2 -8721.166} C_VEL
LIN {X 0,Y 445.911,Z 609.444,A -85,B 0,C 180,E1 -8722.074,E2 -8722.074} C_VEL
LIN {X 0,Y 445.776,Z 614.646,A -85,B 0,C 180,E1 -8722.983,E2 -8722.983} C_VEL
LIN {X 0,Y 445.573,Z 619.935,A -85,B 0,C 180,E1 -8724.116,E2 -8724.116} C_VEL
LIN {X 0,Y 445.451,Z 624.843,A -85,B 0,C 180,E1 -8725.476,E2 -8725.476} C_VEL
LIN {X 0,Y 445.453,Z 627.24,A -85,B 0,C 180,E1 -8726.382,E2 -8726.382} C_VEL
LIN {X 0,Y 445.459,Z 629.065,A -85,B 0,C 180,E1 -8727.288,E2 -8727.288} C_VEL
LIN {X 0,Y 445.399,Z 630.368,A -85,B 0,C 180,E1 -8728.192,E2 -8728.192} C_VEL
LIN {X 0,Y 445.393,Z 631.18,A -85,B 0,C 180,E1 -8729.096,E2 -8729.096} C_VEL
LIN {X 0,Y 445.397,Z 631.452,A -85,B 0,C 180,E1 -8730,E2 -8730} C_VEL
LIN {X 0,Y 445.393,Z 631.136,A -85,B 0,C 180,E1 -8730.905,E2 -8730.905} C_VEL
LIN {X 0,Y 445.399,Z 630.318,A -85,B 0,C 180,E1 -8731.809,E2 -8731.809} C_VEL
LIN {X 0,Y 445.46,Z 629.011,A -85,B 0,C 180,E1 -8732.713,E2 -8732.713} C_VEL
LIN {X 0,Y 445.43,Z 625.982,A -85,B 0,C 180,E1 -8734.072,E2 -8734.072} C_VEL
LIN {X 0,Y 445.524,Z 623.233,A -85,B 0,C 180,E1 -8734.978,E2 -8734.978} C_VEL
LIN {X 0,Y 445.645,Z 617.87,A -85,B 0,C 180,E1 -8736.338,E2 -8736.338} C_VEL
LIN {X 0,Y 445.855,Z 610.806,A -85,B 0,C 180,E1 -8737.7,E2 -8737.7} C_VEL
LIN {X 0,Y 446.14,Z 603.148,A -85,B 0,C 180,E1 -8738.836,E2 -8738.836} C_VEL
LIN {X 0,Y 446.514,Z 595.632,A -85,B 0,C 180,E1 -8739.742,E2 -8739.742} C_VEL
LIN {X 0,Y 446.874,Z 587.638,A -85,B 0,C 180,E1 -8740.535,E2 -8740.535} C_VEL
LIN {X 0,Y 447.29,Z 577.807,A -85,B 0,C 180,E1 -8741.327,E2 -8741.327} C_VEL
LIN {X 0,Y 447.45,Z 568.007,A -85,B 0,C 180,E1 -8741.939,E2 -8741.939} C_VEL
LIN {X 0,Y 446.524,Z 556.911,A -85,B 0,C 180,E1 -8742.486,E2 -8742.486} C_VEL
LIN {X 0,Y 445.58,Z 548.846,A -85,B 0,C 180,E1 -8742.815,E2 -8742.815} C_VEL
LIN {X 0,Y 445.774,Z 540.441,A -85,B 0,C 180,E1 -8745.906,E2 -8745.906} C_VEL
LIN {X 0,Y 446.016,Z 531.398,A -85,B 0,C 180,E1 -8749.324,E2 -8749.324} C_VEL
LIN {X 0,Y 446.283,Z 524.058,A -85,B 0,C 180,E1 -8752.207,E2 -8752.207} C_VEL
LIN {X 0,Y 446.648,Z 516.936,A -85,B 0,C 180,E1 -8755.141,E2 -8755.141} C_VEL
LIN {X 0,Y 447.173,Z 509.659,A -85,B 0,C 180,E1 -8758.343,E2 -8758.343} C_VEL
LIN {X 0,Y 447.737,Z 503.734,A -85,B 0,C 180,E1 -8761.198,E2 -8761.198} C_VEL
LIN {X 0,Y 447.983,Z 499.819,A -85,B 0,C 180,E1 -8763.305,E2 -8763.305} C_VEL
LIN {X 0,Y 447.593,Z 496.304,A -85,B 0,C 180,E1 -8765.519,E2 -8765.519} C_VEL
LIN {X 0,Y 446.991,Z 492.849,A -85,B 0,C 180,E1 -8768.173,E2 -8768.173} C_VEL
LIN {X 0,Y 446.502,Z 490.155,A -85,B 0,C 180,E1 -8770.929,E2 -8770.929} C_VEL
LIN {X 0,Y 446.434,Z 489.793,A -85,B 0,C 180,E1 -8771.391,E2 -8771.391} C_VEL
LIN {X 0,Y 446.457,Z 489.687,A -85,B 0,C 180,E1 -8774.897,E2 -8774.897} C_VEL
LIN {X 0,Y 446.439,Z 489.689,A -85,B 0,C 180,E1 -8777.723,E2 -8777.723} C_VEL
LIN {X 0,Y 446.458,Z 489.687,A -85,B 0,C 180,E1 -8780.975,E2 -8780.975} C_VEL
LIN {X 0,Y 446.42,Z 489.693,A -85,B 0,C 180,E1 -8784.374,E2 -8784.374} C_VEL
LIN {X 0,Y 446.574,Z 490.918,A -85,B 0,C 180,E1 -8786.577,E2 -8786.577} C_VEL
LIN {X 0,Y 446.589,Z 492.509,A -85,B 0,C 180,E1 -8788.713,E2 -8788.713} C_VEL
LIN {X 0,Y 446.37,Z 495.209,A -85,B 0,C 180,E1 -8791.85,E2 -8791.85} C_VEL
LIN {X 0,Y 446.158,Z 498.049,A -85,B 0,C 180,E1 -8794.83,E2 -8794.83} C_VEL
LIN {X 0,Y 445.962,Z 501.711,A -85,B 0,C 180,E1 -8798.403,E2 -8798.403} C_VEL
LIN {X 0,Y 445.833,Z 505.21,A -85,B 0,C 180,E1 -8801.623,E2 -8801.623} C_VEL
LIN {X 0,Y 445.772,Z 508.416,A -85,B 0,C 180,E1 -8804.454,E2 -8804.454} C_VEL
LIN {X 0,Y 445.696,Z 511.792,A -85,B 0,C 180,E1 -8807.339,E2 -8807.339} C_VEL
LIN {X 0,Y 447.785,Z 522.563,A -85,B 0,C 180,E1 -8807.866,E2 -8807.866} C_VEL
LIN {X 0,Y 448.036,Z 529.299,A -85,B 0,C 180,E1 -8808.234,E2 -8808.234} C_VEL
LIN {X 0,Y 447.608,Z 539.3,A -85,B 0,C 180,E1 -8808.911,E2 -8808.911} C_VEL
LIN {X 0,Y 447.287,Z 547.301,A -85,B 0,C 180,E1 -8809.59,E2 -8809.59} C_VEL
LIN {X 0,Y 446.995,Z 553.962,A -85,B 0,C 180,E1 -8810.269,E2 -8810.269} C_VEL
LIN {X 0,Y 446.661,Z 561.325,A -85,B 0,C 180,E1 -8811.175,E2 -8811.175} C_VEL
LIN {X 0,Y 446.328,Z 567.419,A -85,B 0,C 180,E1 -8812.081,E2 -8812.081} C_VEL
LIN {X 0,Y 446.164,Z 572.166,A -85,B 0,C 180,E1 -8812.925,E2 -8812.925} C_VEL
LIN {X 0,Y 446.057,Z 575.76,A -85,B 0,C 180,E1 -8813.668,E2 -8813.668} C_VEL
LIN {X 0,Y 445.702,Z 579.464,A -85,B 0,C 180,E1 -8814.571,E2 -8814.571} C_VEL
LIN {X 0,Y 445.788,Z 582.447,A -85,B 0,C 180,E1 -8815.479,E2 -8815.479} C_VEL
LIN {X 0,Y 445.63,Z 584.771,A -85,B 0,C 180,E1 -8816.383,E2 -8816.383} C_VEL
LIN {X 0,Y 445.532,Z 586.532,A -85,B 0,C 180,E1 -8817.288,E2 -8817.288} C_VEL
LIN {X 0,Y 445.501,Z 587.781,A -85,B 0,C 180,E1 -8818.192,E2 -8818.192} C_VEL
LIN {X 0,Y 445.427,Z 588.548,A -85,B 0,C 180,E1 -8819.096,E2 -8819.096} C_VEL
LIN {X 0,Y 445.399,Z 588.808,A -85,B 0,C 180,E1 -8820,E2 -8820} C_VEL
LIN {X 0,Y 445.411,Z 588.471,A -85,B 0,C 180,E1 -8820.904,E2 -8820.904} C_VEL
LIN {X 0,Y 445.458,Z 587.637,A -85,B 0,C 180,E1 -8821.808,E2 -8821.808} C_VEL
LIN {X 0,Y 445.519,Z 586.312,A -85,B 0,C 180,E1 -8822.713,E2 -8822.713} C_VEL
LIN {X 0,Y 445.68,Z 583.294,A -85,B 0,C 180,E1 -8824.069,E2 -8824.069} C_VEL
LIN {X 0,Y 445.69,Z 578.993,A -85,B 0,C 180,E1 -8825.429,E2 -8825.429} C_VEL
LIN {X 0,Y 446.096,Z 573.397,A -85,B 0,C 180,E1 -8826.722,E2 -8826.722} C_VEL
LIN {X 0,Y 446.171,Z 568.131,A -85,B 0,C 180,E1 -8827.695,E2 -8827.695} C_VEL
LIN {X 0,Y 446.395,Z 562.181,A -85,B 0,C 180,E1 -8828.602,E2 -8828.602} C_VEL
LIN {X 0,Y 446.745,Z 554.962,A -85,B 0,C 180,E1 -8829.508,E2 -8829.508} C_VEL
LIN {X 0,Y 447.077,Z 547.3,A -85,B 0,C 180,E1 -8830.301,E2 -8830.301} C_VEL
LIN {X 0,Y 447.411,Z 539.307,A -85,B 0,C 180,E1 -8830.98,E2 -8830.98} C_VEL
LIN {X 0,Y 447.745,Z 531.109,A -85,B 0,C 180,E1 -8831.545,E2 -8831.545} C_VEL
LIN {X 0,Y 447.682,Z 522.624,A -85,B 0,C 180,E1 -8832.018,E2 -8832.018} C_VEL
LIN {X 0,Y 445.991,Z 512.369,A -85,B 0,C 180,E1 -8832.491,E2 -8832.491} C_VEL
LIN {X 0,Y 445.573,Z 510.003,A -85,B 0,C 180,E1 -8832.599,E2 -8832.599} C_VEL
LIN {X 0,Y 445.616,Z 505.467,A -85,B 0,C 180,E1 -8835.832,E2 -8835.832} C_VEL
LIN {X 0,Y 445.642,Z 500.645,A -85,B 0,C 180,E1 -8839.341,E2 -8839.341} C_VEL
LIN {X 0,Y 445.677,Z 496.725,A -85,B 0,C 180,E1 -8842.239,E2 -8842.239} C_VEL
LIN {X 0,Y 445.8,Z 492.792,A -85,B 0,C 180,E1 -8845.192,E2 -8845.192} C_VEL
LIN {X 0,Y 445.986,Z 490.532,A -85,B 0,C 180,E1 -8846.971,E2 -8846.971} C_VEL
LIN {X 0,Y 446.068,Z 495.683,A -85,B 0,C 180,E1 -8849.237,E2 -8849.237} C_VEL
LIN {X 0,Y 446.014,Z 502.804,A -85,B 0,C 180,E1 -8852.395,E2 -8852.395} C_VEL
LIN {X 0,Y 445.947,Z 508.518,A -85,B 0,C 180,E1 -8854.964,E2 -8854.964} C_VEL
LIN {X 0,Y 445.808,Z 516.354,A -85,B 0,C 180,E1 -8858.513,E2 -8858.513} C_VEL
LIN {X 0,Y 445.693,Z 522.864,A -85,B 0,C 180,E1 -8861.475,E2 -8861.475} C_VEL
LIN {X 0,Y 445.701,Z 527.154,A -85,B 0,C 180,E1 -8863.361,E2 -8863.361} C_VEL
LIN {X 0,Y 447.291,Z 536.875,A -85,B 0,C 180,E1 -8863.737,E2 -8863.737} C_VEL
LIN {X 0,Y 447.948,Z 543,A -85,B 0,C 180,E1 -8864.035,E2 -8864.035} C_VEL
LIN {X 0,Y 447.745,Z 551.3,A -85,B 0,C 180,E1 -8864.504,E2 -8864.504} C_VEL
LIN {X 0,Y 447.397,Z 558.657,A -85,B 0,C 180,E1 -8865.017,E2 -8865.017} C_VEL
LIN {X 0,Y 447.051,Z 567.239,A -85,B 0,C 180,E1 -8865.764,E2 -8865.764} C_VEL
LIN {X 0,Y 446.69,Z 574.83,A -85,B 0,C 180,E1 -8866.577,E2 -8866.577} C_VEL
LIN {X 0,Y 446.314,Z 582.651,A -85,B 0,C 180,E1 -8867.603,E2 -8867.603} C_VEL
LIN {X 0,Y 445.925,Z 590.227,A -85,B 0,C 180,E1 -8868.894,E2 -8868.894} C_VEL
LIN {X 0,Y 445.779,Z 594.229,A -85,B 0,C 180,E1 -8869.729,E2 -8869.729} C_VEL
LIN {X 0,Y 445.613,Z 598.67,A -85,B 0,C 180,E1 -8870.886,E2 -8870.886} C_VEL
LIN {X 0,Y 445.5,Z 602.15,A -85,B 0,C 180,E1 -8872.072,E2 -8872.072} C_VEL
LIN {X 0,Y 445.383,Z 604.476,A -85,B 0,C 180,E1 -8873.156,E2 -8873.156} C_VEL
LIN {X 0,Y 445.291,Z 606.063,A -85,B 0,C 180,E1 -8874.269,E2 -8874.269} C_VEL
LIN {X 0,Y 445.246,Z 606.876,A -85,B 0,C 180,E1 -8875.372,E2 -8875.372} C_VEL
LIN {X 0,Y 445.215,Z 606.837,A -85,B 0,C 180,E1 -8876.787,E2 -8876.787} C_VEL
LIN {X 0,Y 445.34,Z 605.254,A -85,B 0,C 180,E1 -8878.45,E2 -8878.45} C_VEL
LIN {X 0,Y 445.446,Z 602.904,A -85,B 0,C 180,E1 -8879.676,E2 -8879.676} C_VEL
LIN {X 0,Y 445.536,Z 600.111,A -85,B 0,C 180,E1 -8880.725,E2 -8880.725} C_VEL
LIN {X 0,Y 445.717,Z 595.516,A -85,B 0,C 180,E1 -8882.006,E2 -8882.006} C_VEL
LIN {X 0,Y 445.972,Z 589.43,A -85,B 0,C 180,E1 -8883.312,E2 -8883.312} C_VEL
LIN {X 0,Y 446.335,Z 581.621,A -85,B 0,C 180,E1 -8884.59,E2 -8884.59} C_VEL
LIN {X 0,Y 446.638,Z 574.693,A -85,B 0,C 180,E1 -8885.492,E2 -8885.492} C_VEL
LIN {X 0,Y 447,Z 567.734,A -85,B 0,C 180,E1 -8886.24,E2 -8886.24} C_VEL
LIN {X 0,Y 447.239,Z 560.779,A -85,B 0,C 180,E1 -8886.867,E2 -8886.867} C_VEL
LIN {X 0,Y 447.609,Z 553.254,A -85,B 0,C 180,E1 -8887.424,E2 -8887.424} C_VEL
LIN {X 0,Y 447.874,Z 543.641,A -85,B 0,C 180,E1 -8887.987,E2 -8887.987} C_VEL
LIN {X 0,Y 446.928,Z 535.458,A -85,B 0,C 180,E1 -8888.381,E2 -8888.381} C_VEL
LIN {X 0,Y 445.523,Z 527.038,A -85,B 0,C 180,E1 -8888.726,E2 -8888.726} C_VEL
LIN {X 0,Y 445.593,Z 521.345,A -85,B 0,C 180,E1 -8891.522,E2 -8891.522} C_VEL
LIN {X 0,Y 444.972,Z 519.914,A -85,B 0,C 180,E1 -8892.254,E2 -8892.254} C_VEL
LIN {X 0,Y 442.152,Z 517.732,A -85,B 0,C 180,E1 -8893.449,E2 -8893.449} C_VEL
LIN {X 0,Y 439.744,Z 515.981,A -85,B 0,C 180,E1 -8894.414,E2 -8894.414} C_VEL
LIN {X 0,Y 438.709,Z 514.57,A -85,B 0,C 180,E1 -8895.157,E2 -8895.157} C_VEL
LIN {X 0,Y 438.625,Z 514.073,A -85,B 0,C 180,E1 -8895.408,E2 -8895.408} C_VEL
LIN {X 0,Y 438.819,Z 508.916,A -85,B 0,C 180,E1 -8897.982,E2 -8897.982} C_VEL
LIN {X 0,Y 438.872,Z 503.19,A -85,B 0,C 180,E1 -8900.785,E2 -8900.785} C_VEL
LIN {X 0,Y 438.971,Z 497.48,A -85,B 0,C 180,E1 -8903.565,E2 -8903.565} C_VEL
LIN {X 0,Y 439.126,Z 493.731,A -85,B 0,C 180,E1 -8905.41,E2 -8905.41} C_VEL
LIN {X 0,Y 439.058,Z 490.61,A -85,B 0,C 180,E1 -8907.018,E2 -8907.018} C_VEL
LIN {X 0,Y 439.565,Z 490.544,A -85,B 0,C 180,E1 -8909.083,E2 -8909.083} C_VEL
LIN {X 0,Y 439.758,Z 490.521,A -85,B 0,C 180,E1 -8910,E2 -8910} C_VEL
LIN {X 0,Y 439.657,Z 490.534,A -85,B 0,C 180,E1 -8912.748,E2 -8912.748} C_VEL
LIN {X 0,Y 439.621,Z 490.54,A -85,B 0,C 180,E1 -8916.425,E2 -8916.425} C_VEL
LIN {X 0,Y 439.5,Z 490.55,A -85,B 0,C 180,E1 -8919.201,E2 -8919.201} C_VEL
LIN {X 0,Y 439.467,Z 490.556,A -85,B 0,C 180,E1 -8922.937,E2 -8922.937} C_VEL
LIN {X 0,Y 439.448,Z 490.56,A -85,B 0,C 180,E1 -8926.348,E2 -8926.348} C_VEL
LIN {X 0,Y 439.403,Z 490.565,A -85,B 0,C 180,E1 -8929.626,E2 -8929.626} C_VEL
LIN {X 0,Y 439.366,Z 490.57,A -85,B 0,C 180,E1 -8932.575,E2 -8932.575} C_VEL
LIN {X 0,Y 439.406,Z 490.564,A -85,B 0,C 180,E1 -8935.584,E2 -8935.584} C_VEL
LIN {X 0,Y 439.425,Z 490.563,A -85,B 0,C 180,E1 -8938.672,E2 -8938.672} C_VEL
LIN {X 0,Y 439.374,Z 490.569,A -85,B 0,C 180,E1 -8941.86,E2 -8941.86} C_VEL
LIN {X 0,Y 439.4,Z 490.563,A -85,B 0,C 180,E1 -8945.155,E2 -8945.155} C_VEL
LIN {X 0,Y 439.389,Z 490.566,A -85,B 0,C 180,E1 -8948.594,E2 -8948.594} C_VEL
LIN {X 0,Y 439.388,Z 490.565,A -85,B 0,C 180,E1 -8951.256,E2 -8951.256} C_VEL
LIN {X 0,Y 439.405,Z 490.563,A -85,B 0,C 180,E1 -8954.728,E2 -8954.728} C_VEL
LIN {X 0,Y 439.411,Z 490.565,A -85,B 0,C 180,E1 -8957.797,E2 -8957.797} C_VEL
LIN {X 0,Y 439.449,Z 490.56,A -85,B 0,C 180,E1 -8960.23,E2 -8960.23} C_VEL
LIN {X 0,Y 439.373,Z 490.569,A -85,B 0,C 180,E1 -8963.713,E2 -8963.713} C_VEL
LIN {X 0,Y 439.37,Z 490.567,A -85,B 0,C 180,E1 -8967.054,E2 -8967.054} C_VEL
LIN {X 0,Y 439.38,Z 490.568,A -85,B 0,C 180,E1 -8970.274,E2 -8970.274} C_VEL
LIN {X 0,Y 439.428,Z 490.562,A -85,B 0,C 180,E1 -8973.396,E2 -8973.396} C_VEL
LIN {X 0,Y 439.385,Z 490.568,A -85,B 0,C 180,E1 -8976.429,E2 -8976.429} C_VEL
LIN {X 0,Y 439.387,Z 490.567,A -85,B 0,C 180,E1 -8979.397,E2 -8979.397} C_VEL
LIN {X 0,Y 439.429,Z 490.563,A -85,B 0,C 180,E1 -8982.309,E2 -8982.309} C_VEL
LIN {X 0,Y 439.445,Z 490.559,A -85,B 0,C 180,E1 -8985.174,E2 -8985.174} C_VEL
LIN {X 0,Y 439.505,Z 490.553,A -85,B 0,C 180,E1 -8988.002,E2 -8988.002} C_VEL
LIN {X 0,Y 439.546,Z 490.548,A -85,B 0,C 180,E1 -8991.726,E2 -8991.726} C_VEL
LIN {X 0,Y 439.619,Z 490.537,A -85,B 0,C 180,E1 -8994.496,E2 -8994.496} C_VEL
LIN {X 0,Y 439.634,Z 490.536,A -85,B 0,C 180,E1 -8998.168,E2 -8998.168} C_VEL
LIN {X 0,Y 439.761,Z 490.521,A -85,B 0,C 180,E1 -9000,E2 -9000} C_VEL
LIN {X 0,Y 439.655,Z 490.532,A -85,B 0,C 180,E1 -9002.749,E2 -9002.749} C_VEL
LIN {X 0,Y 439.616,Z 490.537,A -85,B 0,C 180,E1 -9006.425,E2 -9006.425} C_VEL
LIN {X 0,Y 439.498,Z 490.553,A -85,B 0,C 180,E1 -9009.202,E2 -9009.202} C_VEL
LIN {X 0,Y 439.462,Z 490.555,A -85,B 0,C 180,E1 -9012.938,E2 -9012.938} C_VEL
LIN {X 0,Y 439.445,Z 490.559,A -85,B 0,C 180,E1 -9016.349,E2 -9016.349} C_VEL
LIN {X 0,Y 439.4,Z 490.566,A -85,B 0,C 180,E1 -9019.626,E2 -9019.626} C_VEL
LIN {X 0,Y 439.362,Z 490.569,A -85,B 0,C 180,E1 -9022.575,E2 -9022.575} C_VEL
LIN {X 0,Y 439.403,Z 490.566,A -85,B 0,C 180,E1 -9025.585,E2 -9025.585} C_VEL
LIN {X 0,Y 439.422,Z 490.561,A -85,B 0,C 180,E1 -9028.673,E2 -9028.673} C_VEL
LIN {X 0,Y 439.38,Z 490.568,A -85,B 0,C 180,E1 -9032.033,E2 -9032.033} C_VEL
LIN {X 0,Y 439.394,Z 490.566,A -85,B 0,C 180,E1 -9035.341,E2 -9035.341} C_VEL
LIN {X 0,Y 439.386,Z 490.565,A -85,B 0,C 180,E1 -9038.595,E2 -9038.595} C_VEL
LIN {X 0,Y 439.387,Z 490.567,A -85,B 0,C 180,E1 -9041.257,E2 -9041.257} C_VEL
LIN {X 0,Y 439.403,Z 490.563,A -85,B 0,C 180,E1 -9044.729,E2 -9044.729} C_VEL
LIN {X 0,Y 439.395,Z 490.566,A -85,B 0,C 180,E1 -9047.796,E2 -9047.796} C_VEL
LIN {X 0,Y 439.45,Z 490.557,A -85,B 0,C 180,E1 -9050.231,E2 -9050.231} C_VEL
LIN {X 0,Y 439.384,Z 490.569,A -85,B 0,C 180,E1 -9053.714,E2 -9053.714} C_VEL
LIN {X 0,Y 439.448,Z 490.674,A -85,B 0,C 180,E1 -9054.65,E2 -9054.65} C_VEL
LIN {X 0,Y 440.709,Z 497.778,A -85,B 0,C 180,E1 -9057.692,E2 -9057.692} C_VEL
LIN {X 0,Y 440.777,Z 502.057,A -85,B 0,C 180,E1 -9059.43,E2 -9059.43} C_VEL
LIN {X 0,Y 440.266,Z 509.703,A -85,B 0,C 180,E1 -9062.424,E2 -9062.424} C_VEL
LIN {X 0,Y 439.746,Z 518.124,A -85,B 0,C 180,E1 -9065.64,E2 -9065.64} C_VEL
LIN {X 0,Y 439.347,Z 526.859,A -85,B 0,C 180,E1 -9068.905,E2 -9068.905} C_VEL
LIN {X 0,Y 439.01,Z 534.783,A -85,B 0,C 180,E1 -9071.81,E2 -9071.81} C_VEL
LIN {X 0,Y 438.721,Z 544.009,A -85,B 0,C 180,E1 -9075.149,E2 -9075.149} C_VEL
LIN {X 0,Y 438.611,Z 549.872,A -85,B 0,C 180,E1 -9077.197,E2 -9077.197} C_VEL
LIN {X 0,Y 439.855,Z 561.793,A -85,B 0,C 180,E1 -9077.654,E2 -9077.654} C_VEL
LIN {X 0,Y 440.44,Z 570.983,A -85,B 0,C 180,E1 -9078.145,E2 -9078.145} C_VEL
LIN {X 0,Y 440.09,Z 581.164,A -85,B 0,C 180,E1 -9078.836,E2 -9078.836} C_VEL
LIN {X 0,Y 439.695,Z 589.322,A -85,B 0,C 180,E1 -9079.525,E2 -9079.525} C_VEL
LIN {X 0,Y 439.303,Z 598.089,A -85,B 0,C 180,E1 -9080.446,E2 -9080.446} C_VEL
LIN {X 0,Y 438.968,Z 605.996,A -85,B 0,C 180,E1 -9081.484,E2 -9081.484} C_VEL
LIN {X 0,Y 438.716,Z 613.001,A -85,B 0,C 180,E1 -9082.637,E2 -9082.637} C_VEL
LIN {X 0,Y 438.496,Z 618.749,A -85,B 0,C 180,E1 -9083.838,E2 -9083.838} C_VEL
LIN {X 0,Y 438.456,Z 622.929,A -85,B 0,C 180,E1 -9084.943,E2 -9084.943} C_VEL
LIN {X 0,Y 438.352,Z 626.857,A -85,B 0,C 180,E1 -9086.324,E2 -9086.324} C_VEL
LIN {X 0,Y 438.387,Z 628.704,A -85,B 0,C 180,E1 -9087.244,E2 -9087.244} C_VEL
LIN {X 0,Y 438.318,Z 630.02,A -85,B 0,C 180,E1 -9088.163,E2 -9088.163} C_VEL
LIN {X 0,Y 438.303,Z 630.836,A -85,B 0,C 180,E1 -9089.082,E2 -9089.082} C_VEL
LIN {X 0,Y 438.318,Z 631.102,A -85,B 0,C 180,E1 -9090,E2 -9090} C_VEL
LIN {X 0,Y 438.303,Z 630.826,A -85,B 0,C 180,E1 -9090.919,E2 -9090.919} C_VEL
LIN {X 0,Y 438.319,Z 629.991,A -85,B 0,C 180,E1 -9091.838,E2 -9091.838} C_VEL
LIN {X 0,Y 438.388,Z 628.695,A -85,B 0,C 180,E1 -9092.757,E2 -9092.757} C_VEL
LIN {X 0,Y 438.341,Z 625.666,A -85,B 0,C 180,E1 -9094.138,E2 -9094.138} C_VEL
LIN {X 0,Y 438.457,Z 622.928,A -85,B 0,C 180,E1 -9095.058,E2 -9095.058} C_VEL
LIN {X 0,Y 438.521,Z 618.633,A -85,B 0,C 180,E1 -9096.193,E2 -9096.193} C_VEL
LIN {X 0,Y 438.717,Z 613.03,A -85,B 0,C 180,E1 -9097.363,E2 -9097.363} C_VEL
LIN {X 0,Y 438.987,Z 606.192,A -85,B 0,C 180,E1 -9098.517,E2 -9098.517} C_VEL
LIN {X 0,Y 439.385,Z 597.508,A -85,B 0,C 180,E1 -9099.669,E2 -9099.669} C_VEL
LIN {X 0,Y 439.776,Z 589.994,A -85,B 0,C 180,E1 -9100.474,E2 -9100.474} C_VEL
LIN {X 0,Y 440.109,Z 582.244,A -85,B 0,C 180,E1 -9101.165,E2 -9101.165} C_VEL
LIN {X 0,Y 440.53,Z 572.641,A -85,B 0,C 180,E1 -9101.853,E2 -9101.853} C_VEL
LIN {X 0,Y 440.243,Z 565.884,A -85,B 0,C 180,E1 -9102.262,E2 -9102.262} C_VEL
LIN {X 0,Y 439.438,Z 555.589,A -85,B 0,C 180,E1 -9102.765,E2 -9102.765} C_VEL
LIN {X 0,Y 438.513,Z 548.478,A -85,B 0,C 180,E1 -9103.055,E2 -9103.055} C_VEL
LIN {X 0,Y 438.711,Z 540.605,A -85,B 0,C 180,E1 -9106.017,E2 -9106.017} C_VEL
LIN {X 0,Y 438.943,Z 532.49,A -85,B 0,C 180,E1 -9109.151,E2 -9109.151} C_VEL
LIN {X 0,Y 439.183,Z 525.74,A -85,B 0,C 180,E1 -9111.853,E2 -9111.853} C_VEL
LIN {X 0,Y 439.62,Z 518.086,A -85,B 0,C 180,E1 -9115.065,E2 -9115.065} C_VEL
LIN {X 0,Y 440.102,Z 511.359,A -85,B 0,C 180,E1 -9118.087,E2 -9118.087} C_VEL
LIN {X 0,Y 440.767,Z 505.007,A -85,B 0,C 180,E1 -9121.213,E2 -9121.213} C_VEL
LIN {X 0,Y 440.954,Z 502.083,A -85,B 0,C 180,E1 -9122.813,E2 -9122.813} C_VEL
LIN {X 0,Y 440.753,Z 498.492,A -85,B 0,C 180,E1 -9125.033,E2 -9125.033} C_VEL
LIN {X 0,Y 440.237,Z 495.376,A -85,B 0,C 180,E1 -9127.347,E2 -9127.347} C_VEL
LIN {X 0,Y 439.778,Z 492.629,A -85,B 0,C 180,E1 -9129.908,E2 -9129.908} C_VEL
LIN {X 0,Y 439.386,Z 490.581,A -85,B 0,C 180,E1 -9132.628,E2 -9132.628} C_VEL
LIN {X 0,Y 439.408,Z 490.566,A -85,B 0,C 180,E1 -9135.272,E2 -9135.272} C_VEL
LIN {X 0,Y 439.392,Z 490.568,A -85,B 0,C 180,E1 -9138.743,E2 -9138.743} C_VEL
LIN {X 0,Y 439.379,Z 490.569,A -85,B 0,C 180,E1 -9141.608,E2 -9141.608} C_VEL
LIN {X 0,Y 439.376,Z 490.57,A -85,B 0,C 180,E1 -9143.713,E2 -9143.713} C_VEL
LIN {X 0,Y 439.575,Z 491.969,A -85,B 0,C 180,E1 -9146.242,E2 -9146.242} C_VEL
LIN {X 0,Y 439.604,Z 493.289,A -85,B 0,C 180,E1 -9148.158,E2 -9148.158} C_VEL
LIN {X 0,Y 439.495,Z 494.963,A -85,B 0,C 180,E1 -9150.283,E2 -9150.283} C_VEL
LIN {X 0,Y 439.207,Z 497.949,A -85,B 0,C 180,E1 -9153.649,E2 -9153.649} C_VEL
LIN {X 0,Y 439.001,Z 500.613,A -85,B 0,C 180,E1 -9156.408,E2 -9156.408} C_VEL
LIN {X 0,Y 438.879,Z 503.651,A -85,B 0,C 180,E1 -9159.372,E2 -9159.372} C_VEL
LIN {X 0,Y 438.739,Z 506.785,A -85,B 0,C 180,E1 -9162.281,E2 -9162.281} C_VEL
LIN {X 0,Y 438.652,Z 509.996,A -85,B 0,C 180,E1 -9165.147,E2 -9165.147} C_VEL
LIN {X 0,Y 438.661,Z 512.391,A -85,B 0,C 180,E1 -9167.097,E2 -9167.097} C_VEL
LIN {X 0,Y 440.788,Z 522.754,A -85,B 0,C 180,E1 -9167.623,E2 -9167.623} C_VEL
LIN {X 0,Y 441.184,Z 528.887,A -85,B 0,C 180,E1 -9167.966,E2 -9167.966} C_VEL
LIN {X 0,Y 440.708,Z 540.088,A -85,B 0,C 180,E1 -9168.735,E2 -9168.735} C_VEL
LIN {X 0,Y 440.342,Z 548.014,A -85,B 0,C 180,E1 -9169.424,E2 -9169.424} C_VEL
LIN {X 0,Y 440.037,Z 554.617,A -85,B 0,C 180,E1 -9170.114,E2 -9170.114} C_VEL
LIN {X 0,Y 439.69,Z 561.934,A -85,B 0,C 180,E1 -9171.034,E2 -9171.034} C_VEL
LIN {X 0,Y 439.326,Z 567.979,A -85,B 0,C 180,E1 -9171.954,E2 -9171.954} C_VEL
LIN {X 0,Y 439.141,Z 572.941,A -85,B 0,C 180,E1 -9172.864,E2 -9172.864} C_VEL
LIN {X 0,Y 438.833,Z 578.134,A -85,B 0,C 180,E1 -9174.025,E2 -9174.025} C_VEL
LIN {X 0,Y 438.662,Z 581.403,A -85,B 0,C 180,E1 -9174.945,E2 -9174.945} C_VEL
LIN {X 0,Y 438.651,Z 584.041,A -85,B 0,C 180,E1 -9175.866,E2 -9175.866} C_VEL
LIN {X 0,Y 438.461,Z 586.926,A -85,B 0,C 180,E1 -9177.244,E2 -9177.244} C_VEL
LIN {X 0,Y 438.415,Z 588.16,A -85,B 0,C 180,E1 -9178.163,E2 -9178.163} C_VEL
LIN {X 0,Y 438.337,Z 588.909,A -85,B 0,C 180,E1 -9179.081,E2 -9179.081} C_VEL
LIN {X 0,Y 438.32,Z 589.156,A -85,B 0,C 180,E1 -9180,E2 -9180} C_VEL
LIN {X 0,Y 438.321,Z 588.806,A -85,B 0,C 180,E1 -9180.919,E2 -9180.919} C_VEL
LIN {X 0,Y 438.375,Z 587.946,A -85,B 0,C 180,E1 -9181.838,E2 -9181.838} C_VEL
LIN {X 0,Y 438.448,Z 586.598,A -85,B 0,C 180,E1 -9182.756,E2 -9182.756} C_VEL
LIN {X 0,Y 438.6,Z 583.543,A -85,B 0,C 180,E1 -9184.135,E2 -9184.135} C_VEL
LIN {X 0,Y 438.646,Z 579.206,A -85,B 0,C 180,E1 -9185.517,E2 -9185.517} C_VEL
LIN {X 0,Y 439.029,Z 574.043,A -85,B 0,C 180,E1 -9186.733,E2 -9186.733} C_VEL
LIN {X 0,Y 439.129,Z 568.23,A -85,B 0,C 180,E1 -9187.819,E2 -9187.819} C_VEL
LIN {X 0,Y 439.373,Z 562.23,A -85,B 0,C 180,E1 -9188.74,E2 -9188.74} C_VEL
LIN {X 0,Y 439.752,Z 554.953,A -85,B 0,C 180,E1 -9189.66,E2 -9189.66} C_VEL
LIN {X 0,Y 440.092,Z 547.228,A -85,B 0,C 180,E1 -9190.466,E2 -9190.466} C_VEL
LIN {X 0,Y 440.44,Z 539.159,A -85,B 0,C 180,E1 -9191.156,E2 -9191.156} C_VEL
LIN {X 0,Y 440.8,Z 529.059,A -85,B 0,C 180,E1 -9191.846,E2 -9191.846} C_VEL
LIN {X 0,Y 440.569,Z 522.451,A -85,B 0,C 180,E1 -9192.205,E2 -9192.205} C_VEL
LIN {X 0,Y 438.497,Z 510.297,A -85,B 0,C 180,E1 -9192.769,E2 -9192.769} C_VEL
LIN {X 0,Y 438.527,Z 505.9,A -85,B 0,C 180,E1 -9195.932,E2 -9195.932} C_VEL
LIN {X 0,Y 438.584,Z 501.686,A -85,B 0,C 180,E1 -9199.014,E2 -9199.014} C_VEL
